// ---- FBs/B_JKS_OldFB/Memory/INDIRECT_FN.TcPOU
FUNCTION_BLOCK INDIRECT_FN
VAR_INPUT
	BOOL_SV_PB: BOOL;		(*SAVE PB (TS)*)
	BOOL_LD_PB: BOOL;			(*LOAD PB (TS)*)
	INT_P_NO: INT;		(*PROGRAM NO (TS) 1~10*)
	INT_D00:INT;
	INT_D01:INT;
	INT_D02:INT;
	INT_D03:INT;
	INT_D04:INT;
	INT_D05:INT;
	INT_D06:INT;
	INT_D07:INT;
	INT_D08:INT;
	INT_D09:INT;
	INT_D10:INT;
	INT_D11:INT;
	INT_D12:INT;
	INT_D13:INT;
	INT_D14:INT;
	INT_D15:INT;
	INT_D16:INT;
	INT_D17:INT;
	INT_D18:INT;
	INT_D19:INT;
	INT_D20:INT;
	INT_D21:INT;
	INT_D22:INT;
	INT_D23:INT;
	INT_D24:INT;
	INT_D25:INT;
	INT_D26:INT;
	INT_D27:INT;
	INT_D28:INT;
	INT_D29:INT;
	INT_D30:INT;
	STG_STG1:STRING;
END_VAR
VAR_OUTPUT
	SV_PB_IND_BOOL:BOOL;
	LD_PB_IND_BOOL:BOOL;
	D00_INT:INT;
	D01_INT:INT;
	D02_INT:INT;
	D03_INT:INT;
	D04_INT:INT;
	D05_INT:INT;
	D06_INT:INT;
	D07_INT:INT;
	D08_INT:INT;
	D09_INT:INT;
	D10_INT:INT;
	D11_INT:INT;
	D12_INT:INT;
	D13_INT:INT;
	D14_INT:INT;
	D15_INT:INT;
	D16_INT:INT;
	D17_INT:INT;
	D18_INT:INT;
	D19_INT:INT;
	D20_INT:INT;
	D21_INT:INT;
	D22_INT:INT;
	D23_INT:INT;
	D24_INT:INT;
	D25_INT:INT;
	D26_INT:INT;
	D27_INT:INT;
	D28_INT:INT;
	D29_INT:INT;
	D30_INT:INT;
	STG1_STG:STRING;
END_VAR
VAR

	P1B: BOOL;
	P2B: BOOL;
	P3B: BOOL;
	P4B: BOOL;
	P5B: BOOL;
	P6B: BOOL;
	P7B: BOOL;
	P8B: BOOL;
	P9B: BOOL;
	P10B: BOOL;
	SV_HR: BOOL;
	SV_T: TON;
	SV_CR: BOOL;
	LD_HR: BOOL;
	LD_CR: BOOL;
	LD_T: TON;
	SV_DF: R_TRIG;
	SV_PLS: BOOL;
	LD_DF: R_TRIG;
	LD_PLS: BOOL;
	ALWAYS_ON: BOOL;
	TPC: TON;
	N0: BOOL;
	TPC1: TON;
	N1: BOOL;
	CNG_P_NO: INT;
	NPC: BOOL;		(*NON PROGRAM CHANGE*)
	PCDF: R_TRIG;
	PCTDF: BOOL;
	PCDFN: F_TRIG;
	PC_PLS: BOOL;
	SVPLS: R_TRIG;
	SV_PB_PLS: BOOL;
	LDPLS: R_TRIG;
	LD_PB_PLS: BOOL;
END_VAR
VAR PERSISTENT
	P01D00:INT;
	P01D01:INT;
	P01D02:INT;
	P01D03:INT;
	P01D04:INT;
	P01D05:INT;
	P01D06:INT;
	P01D07:INT;
	P01D08:INT;
	P01D09:INT;
	P01D10:INT;
	P01D11:INT;
	P01D12:INT;
	P01D13:INT;
	P01D14:INT;
	P01D15:INT;
	P01D16:INT;
	P01D17:INT;
	P01D18:INT;
	P01D19:INT;
	P01D20:INT;
	P01D21:INT;
	P01D22:INT;
	P01D23:INT;
	P01D24:INT;
	P01D25:INT;
	P01D26:INT;
	P01D27:INT;
	P01D28:INT;
	P01D29:INT;
	P01D30:INT;
	P01STG:STRING;
	P02D00:INT;
	P02D01:INT;
	P02D02:INT;
	P02D03:INT;
	P02D04:INT;
	P02D05:INT;
	P02D06:INT;
	P02D07:INT;
	P02D08:INT;
	P02D09:INT;
	P02D10:INT;
	P02D11:INT;
	P02D12:INT;
	P02D13:INT;
	P02D14:INT;
	P02D15:INT;
	P02D16:INT;
	P02D17:INT;
	P02D18:INT;
	P02D19:INT;
	P02D20:INT;
	P02D21:INT;
	P02D22:INT;
	P02D23:INT;
	P02D24:INT;
	P02D25:INT;
	P02D26:INT;
	P02D27:INT;
	P02D28:INT;
	P02D29:INT;
	P02D30:INT;
	P02STG:STRING;
	P03D00:INT;
	P03D01:INT;
	P03D02:INT;
	P03D03:INT;
	P03D04:INT;
	P03D05:INT;
	P03D06:INT;
	P03D07:INT;
	P03D08:INT;
	P03D09:INT;
	P03D10:INT;
	P03D11:INT;
	P03D12:INT;
	P03D13:INT;
	P03D14:INT;
	P03D15:INT;
	P03D16:INT;
	P03D17:INT;
	P03D18:INT;
	P03D19:INT;
	P03D20:INT;
	P03D21:INT;
	P03D22:INT;
	P03D23:INT;
	P03D24:INT;
	P03D25:INT;
	P03D26:INT;
	P03D27:INT;
	P03D28:INT;
	P03D29:INT;
	P03D30:INT;
	P03STG:STRING;
	P04D00:INT;
	P04D01:INT;
	P04D02:INT;
	P04D03:INT;
	P04D04:INT;
	P04D05:INT;
	P04D06:INT;
	P04D07:INT;
	P04D08:INT;
	P04D09:INT;
	P04D10:INT;
	P04D11:INT;
	P04D12:INT;
	P04D13:INT;
	P04D14:INT;
	P04D15:INT;
	P04D16:INT;
	P04D17:INT;
	P04D18:INT;
	P04D19:INT;
	P04D20:INT;
	P04D21:INT;
	P04D22:INT;
	P04D23:INT;
	P04D24:INT;
	P04D25:INT;
	P04D26:INT;
	P04D27:INT;
	P04D28:INT;
	P04D29:INT;
	P04D30:INT;
	P04STG:STRING;
	P05D00:INT;
	P05D01:INT;
	P05D02:INT;
	P05D03:INT;
	P05D04:INT;
	P05D05:INT;
	P05D06:INT;
	P05D07:INT;
	P05D08:INT;
	P05D09:INT;
	P05D10:INT;
	P05D11:INT;
	P05D12:INT;
	P05D13:INT;
	P05D14:INT;
	P05D15:INT;
	P05D16:INT;
	P05D17:INT;
	P05D18:INT;
	P05D19:INT;
	P05D20:INT;
	P05D21:INT;
	P05D22:INT;
	P05D23:INT;
	P05D24:INT;
	P05D25:INT;
	P05D26:INT;
	P05D27:INT;
	P05D28:INT;
	P05D29:INT;
	P05D30:INT;
	P05STG:STRING;
	P06D00:INT;
	P06D01:INT;
	P06D02:INT;
	P06D03:INT;
	P06D04:INT;
	P06D05:INT;
	P06D06:INT;
	P06D07:INT;
	P06D08:INT;
	P06D09:INT;
	P06D10:INT;
	P06D11:INT;
	P06D12:INT;
	P06D13:INT;
	P06D14:INT;
	P06D15:INT;
	P06D16:INT;
	P06D17:INT;
	P06D18:INT;
	P06D19:INT;
	P06D20:INT;
	P06D21:INT;
	P06D22:INT;
	P06D23:INT;
	P06D24:INT;
	P06D25:INT;
	P06D26:INT;
	P06D27:INT;
	P06D28:INT;
	P06D29:INT;
	P06D30:INT;
	P06STG:STRING;
	P07D00:INT;
	P07D01:INT;
	P07D02:INT;
	P07D03:INT;
	P07D04:INT;
	P07D05:INT;
	P07D06:INT;
	P07D07:INT;
	P07D08:INT;
	P07D09:INT;
	P07D10:INT;
	P07D11:INT;
	P07D12:INT;
	P07D13:INT;
	P07D14:INT;
	P07D15:INT;
	P07D16:INT;
	P07D17:INT;
	P07D18:INT;
	P07D19:INT;
	P07D20:INT;
	P07D21:INT;
	P07D22:INT;
	P07D23:INT;
	P07D24:INT;
	P07D25:INT;
	P07D26:INT;
	P07D27:INT;
	P07D28:INT;
	P07D29:INT;
	P07D30:INT;
	P07STG:STRING;
	P08D00:INT;
	P08D01:INT;
	P08D02:INT;
	P08D03:INT;
	P08D04:INT;
	P08D05:INT;
	P08D06:INT;
	P08D07:INT;
	P08D08:INT;
	P08D09:INT;
	P08D10:INT;
	P08D11:INT;
	P08D12:INT;
	P08D13:INT;
	P08D14:INT;
	P08D15:INT;
	P08D16:INT;
	P08D17:INT;
	P08D18:INT;
	P08D19:INT;
	P08D20:INT;
	P08D21:INT;
	P08D22:INT;
	P08D23:INT;
	P08D24:INT;
	P08D25:INT;
	P08D26:INT;
	P08D27:INT;
	P08D28:INT;
	P08D29:INT;
	P08D30:INT;
	P08STG:STRING;
	P09D00:INT;
	P09D01:INT;
	P09D02:INT;
	P09D03:INT;
	P09D04:INT;
	P09D05:INT;
	P09D06:INT;
	P09D07:INT;
	P09D08:INT;
	P09D09:INT;
	P09D10:INT;
	P09D11:INT;
	P09D12:INT;
	P09D13:INT;
	P09D14:INT;
	P09D15:INT;
	P09D16:INT;
	P09D17:INT;
	P09D18:INT;
	P09D19:INT;
	P09D20:INT;
	P09D21:INT;
	P09D22:INT;
	P09D23:INT;
	P09D24:INT;
	P09D25:INT;
	P09D26:INT;
	P09D27:INT;
	P09D28:INT;
	P09D29:INT;
	P09D30:INT;
	P09STG:STRING;
	P10D00:INT;
	P10D01:INT;
	P10D02:INT;
	P10D03:INT;
	P10D04:INT;
	P10D05:INT;
	P10D06:INT;
	P10D07:INT;
	P10D08:INT;
	P10D09:INT;
	P10D10:INT;
	P10D11:INT;
	P10D12:INT;
	P10D13:INT;
	P10D14:INT;
	P10D15:INT;
	P10D16:INT;
	P10D17:INT;
	P10D18:INT;
	P10D19:INT;
	P10D20:INT;
	P10D21:INT;
	P10D22:INT;
	P10D23:INT;
	P10D24:INT;
	P10D25:INT;
	P10D26:INT;
	P10D27:INT;
	P10D28:INT;
	P10D29:INT;
	P10D30:INT;
	P10STG:STRING;

END_VAR
VAR // added by the converter: edge detectors and wires of the graphical bodies
    _w1, _w35, _w68, _w101, _w134, _w167, _w200, _w233, _w266, _w299, _w332, _w365, _w398, _w431, _w464, _w497, _w530, _w563, _w596, _w629, _w662 : BOOL;
    _w2, _w3, _w4, _w5, _w6, _w7, _w8, _w9, _w10, _w11, _w12, _w13, _w14, _w15, _w16, _w17, _w18, _w19, _w20, _w21, _w22, _w23, _w24, _w25, _w26, _w27, _w28, _w29, _w30, _w31, _w32, _w34, _w36, _w37, _w38, _w39, _w40, _w41, _w42, _w43, _w44, _w45, _w46, _w47, _w48, _w49, _w50, _w51, _w52, _w53, _w54, _w55, _w56, _w57, _w58, _w59, _w60, _w61, _w62, _w63, _w64, _w65, _w66, _w69, _w70, _w71, _w72, _w73, _w74, _w75, _w76, _w77, _w78, _w79, _w80, _w81, _w82, _w83, _w84, _w85, _w86, _w87, _w88, _w89, _w90, _w91, _w92, _w93, _w94, _w95, _w96, _w97, _w98, _w99, _w102, _w103, _w104, _w105, _w106, _w107, _w108, _w109, _w110, _w111, _w112, _w113, _w114, _w115, _w116, _w117, _w118, _w119, _w120, _w121, _w122, _w123, _w124, _w125, _w126, _w127, _w128, _w129, _w130, _w131, _w132, _w135, _w136, _w137, _w138, _w139, _w140, _w141, _w142, _w143, _w144, _w145, _w146, _w147, _w148, _w149, _w150, _w151, _w152, _w153, _w154, _w155, _w156, _w157, _w158, _w159, _w160, _w161, _w162, _w163, _w164, _w165, _w168, _w169, _w170, _w171, _w172, _w173, _w174, _w175, _w176, _w177, _w178, _w179, _w180, _w181, _w182, _w183, _w184, _w185, _w186, _w187, _w188, _w189, _w190, _w191, _w192, _w193, _w194, _w195, _w196, _w197, _w198, _w201, _w202, _w203, _w204, _w205, _w206, _w207, _w208, _w209, _w210, _w211, _w212, _w213, _w214, _w215, _w216, _w217, _w218, _w219, _w220, _w221, _w222, _w223, _w224, _w225, _w226, _w227, _w228, _w229, _w230, _w231, _w234, _w235, _w236, _w237, _w238, _w239, _w240, _w241, _w242, _w243, _w244, _w245, _w246, _w247, _w248, _w249, _w250, _w251, _w252, _w253, _w254, _w255, _w256, _w257, _w258, _w259, _w260, _w261, _w262, _w263, _w264, _w267, _w268, _w269, _w270, _w271, _w272, _w273, _w274, _w275, _w276, _w277, _w278, _w279, _w280, _w281, _w282, _w283, _w284, _w285, _w286, _w287, _w288, _w289, _w290, _w291, _w292, _w293, _w294, _w295, _w296, _w297, _w300, _w301, _w302, _w303, _w304, _w305, _w306, _w307, _w308, _w309, _w310, _w311, _w312, _w313, _w314, _w315, _w316, _w317, _w318, _w319, _w320, _w321, _w322, _w323, _w324, _w325, _w326, _w327, _w328, _w329, _w330, _w333, _w334, _w335, _w336, _w337, _w338, _w339, _w340, _w341, _w342, _w343, _w344, _w345, _w346, _w347, _w348, _w349, _w350, _w351, _w352, _w353, _w354, _w355, _w356, _w357, _w358, _w359, _w360, _w361, _w362, _w363, _w366, _w367, _w368, _w369, _w370, _w371, _w372, _w373, _w374, _w375, _w376, _w377, _w378, _w379, _w380, _w381, _w382, _w383, _w384, _w385, _w386, _w387, _w388, _w389, _w390, _w391, _w392, _w393, _w394, _w395, _w396, _w399, _w400, _w401, _w402, _w403, _w404, _w405, _w406, _w407, _w408, _w409, _w410, _w411, _w412, _w413, _w414, _w415, _w416, _w417, _w418, _w419, _w420, _w421, _w422, _w423, _w424, _w425, _w426, _w427, _w428, _w429, _w432, _w433, _w434, _w435, _w436, _w437, _w438, _w439, _w440, _w441, _w442, _w443, _w444, _w445, _w446, _w447, _w448, _w449, _w450, _w451, _w452, _w453, _w454, _w455, _w456, _w457, _w458, _w459, _w460, _w461, _w462, _w465, _w466, _w467, _w468, _w469, _w470, _w471, _w472, _w473, _w474, _w475, _w476, _w477, _w478, _w479, _w480, _w481, _w482, _w483, _w484, _w485, _w486, _w487, _w488, _w489, _w490, _w491, _w492, _w493, _w494, _w495, _w498, _w499, _w500, _w501, _w502, _w503, _w504, _w505, _w506, _w507, _w508, _w509, _w510, _w511, _w512, _w513, _w514, _w515, _w516, _w517, _w518, _w519, _w520, _w521, _w522, _w523, _w524, _w525, _w526, _w527, _w528, _w531, _w532, _w533, _w534, _w535, _w536, _w537, _w538, _w539, _w540, _w541, _w542, _w543, _w544, _w545, _w546, _w547, _w548, _w549, _w550, _w551, _w552, _w553, _w554, _w555, _w556, _w557, _w558, _w559, _w560, _w561, _w564, _w565, _w566, _w567, _w568, _w569, _w570, _w571, _w572, _w573, _w574, _w575, _w576, _w577, _w578, _w579, _w580, _w581, _w582, _w583, _w584, _w585, _w586, _w587, _w588, _w589, _w590, _w591, _w592, _w593, _w594, _w597, _w598, _w599, _w600, _w601, _w602, _w603, _w604, _w605, _w606, _w607, _w608, _w609, _w610, _w611, _w612, _w613, _w614, _w615, _w616, _w617, _w618, _w619, _w620, _w621, _w622, _w623, _w624, _w625, _w626, _w627, _w630, _w631, _w632, _w633, _w634, _w635, _w636, _w637, _w638, _w639, _w640, _w641, _w642, _w643, _w644, _w645, _w646, _w647, _w648, _w649, _w650, _w651, _w652, _w653, _w654, _w655, _w656, _w657, _w658, _w659, _w660, _w663, _w664, _w665, _w666, _w667, _w668, _w669, _w670, _w671, _w672, _w673, _w674, _w675, _w676, _w677, _w678, _w679, _w680, _w681, _w682, _w683, _w684, _w685, _w686, _w687, _w688, _w689, _w690, _w691, _w692, _w693 : INT;
    _w33, _w67, _w100, _w133, _w166, _w199, _w232, _w265, _w298, _w331, _w364, _w397, _w430, _w463, _w496, _w529, _w562, _w595, _w628, _w661, _w694 : STRING;
END_VAR

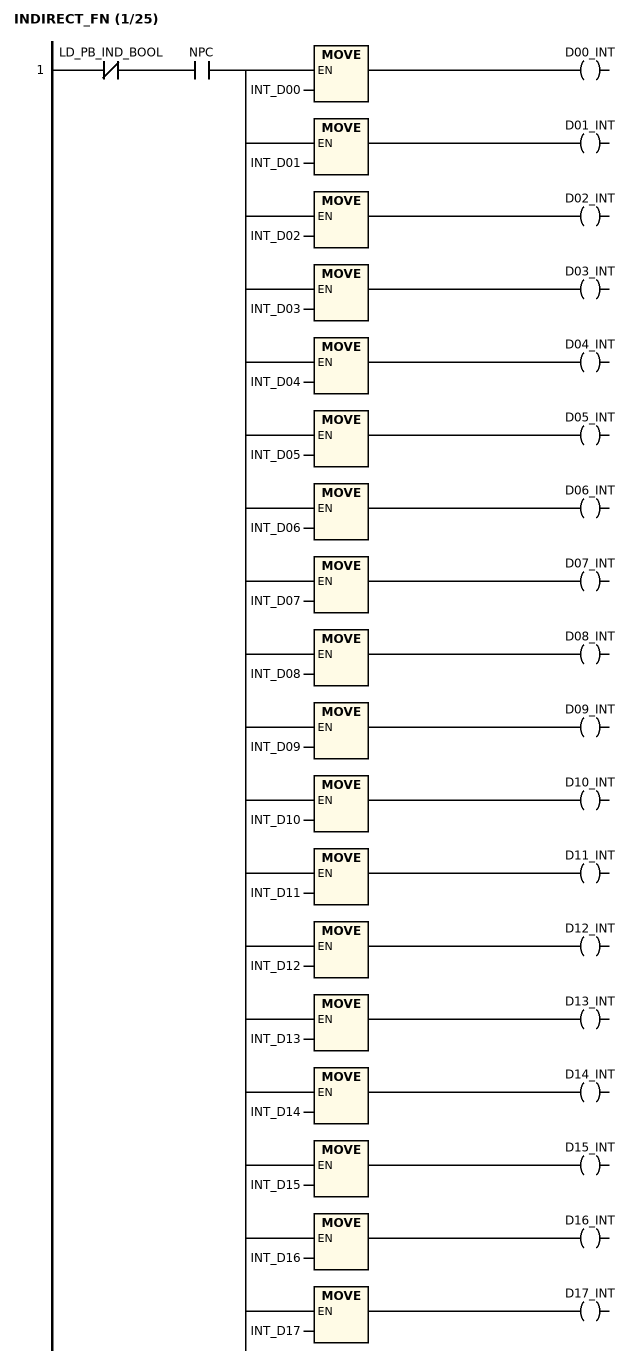
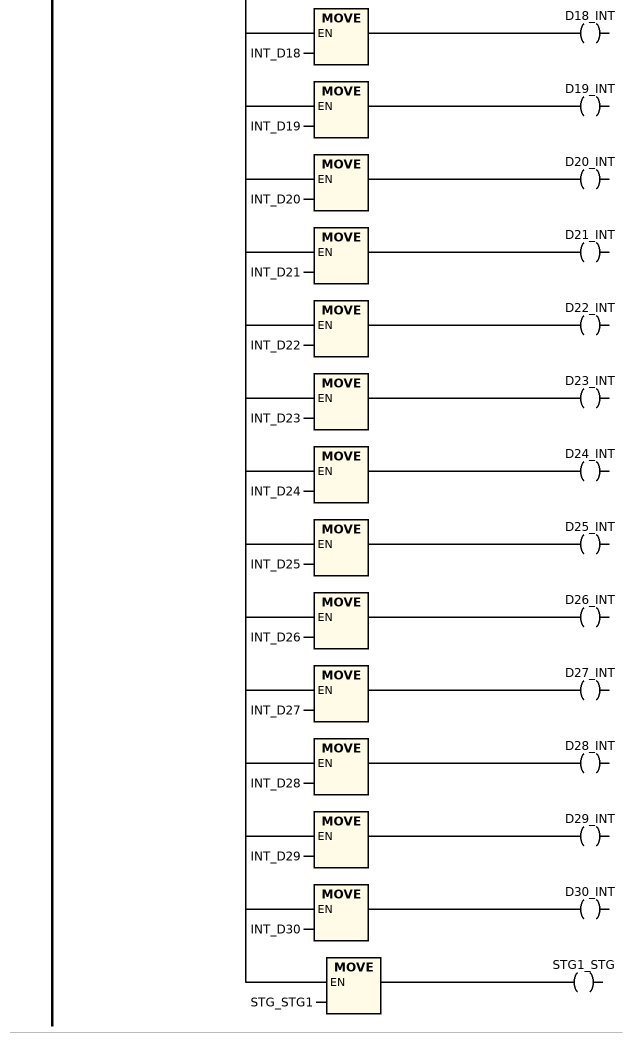
// NETWORK 1
_w1 := NOT LD_PB_IND_BOOL AND NPC;
IF _w1 THEN _w2 := INT_D00; END_IF
D00_INT := _w2;
IF _w1 THEN _w3 := INT_D01; END_IF
D01_INT := _w3;
IF _w1 THEN _w4 := INT_D02; END_IF
D02_INT := _w4;
IF _w1 THEN _w5 := INT_D03; END_IF
D03_INT := _w5;
IF _w1 THEN _w6 := INT_D04; END_IF
D04_INT := _w6;
IF _w1 THEN _w7 := INT_D05; END_IF
D05_INT := _w7;
IF _w1 THEN _w8 := INT_D06; END_IF
D06_INT := _w8;
IF _w1 THEN _w9 := INT_D07; END_IF
D07_INT := _w9;
IF _w1 THEN _w10 := INT_D08; END_IF
D08_INT := _w10;
IF _w1 THEN _w11 := INT_D09; END_IF
D09_INT := _w11;
IF _w1 THEN _w12 := INT_D10; END_IF
D10_INT := _w12;
IF _w1 THEN _w13 := INT_D11; END_IF
D11_INT := _w13;
IF _w1 THEN _w14 := INT_D12; END_IF
D12_INT := _w14;
IF _w1 THEN _w15 := INT_D13; END_IF
D13_INT := _w15;
IF _w1 THEN _w16 := INT_D14; END_IF
D14_INT := _w16;
IF _w1 THEN _w17 := INT_D15; END_IF
D15_INT := _w17;
IF _w1 THEN _w18 := INT_D16; END_IF
D16_INT := _w18;
IF _w1 THEN _w19 := INT_D17; END_IF
D17_INT := _w19;
IF _w1 THEN _w20 := INT_D18; END_IF
D18_INT := _w20;
IF _w1 THEN _w21 := INT_D19; END_IF
D19_INT := _w21;
IF _w1 THEN _w22 := INT_D20; END_IF
D20_INT := _w22;
IF _w1 THEN _w23 := INT_D21; END_IF
D21_INT := _w23;
IF _w1 THEN _w24 := INT_D22; END_IF
D22_INT := _w24;
IF _w1 THEN _w25 := INT_D23; END_IF
D23_INT := _w25;
IF _w1 THEN _w26 := INT_D24; END_IF
D24_INT := _w26;
IF _w1 THEN _w27 := INT_D25; END_IF
D25_INT := _w27;
IF _w1 THEN _w28 := INT_D26; END_IF
D26_INT := _w28;
IF _w1 THEN _w29 := INT_D27; END_IF
D27_INT := _w29;
IF _w1 THEN _w30 := INT_D28; END_IF
D28_INT := _w30;
IF _w1 THEN _w31 := INT_D29; END_IF
D29_INT := _w31;
IF _w1 THEN _w32 := INT_D30; END_IF
D30_INT := _w32;
IF _w1 THEN _w33 := STG_STG1; END_IF
STG1_STG := _w33;

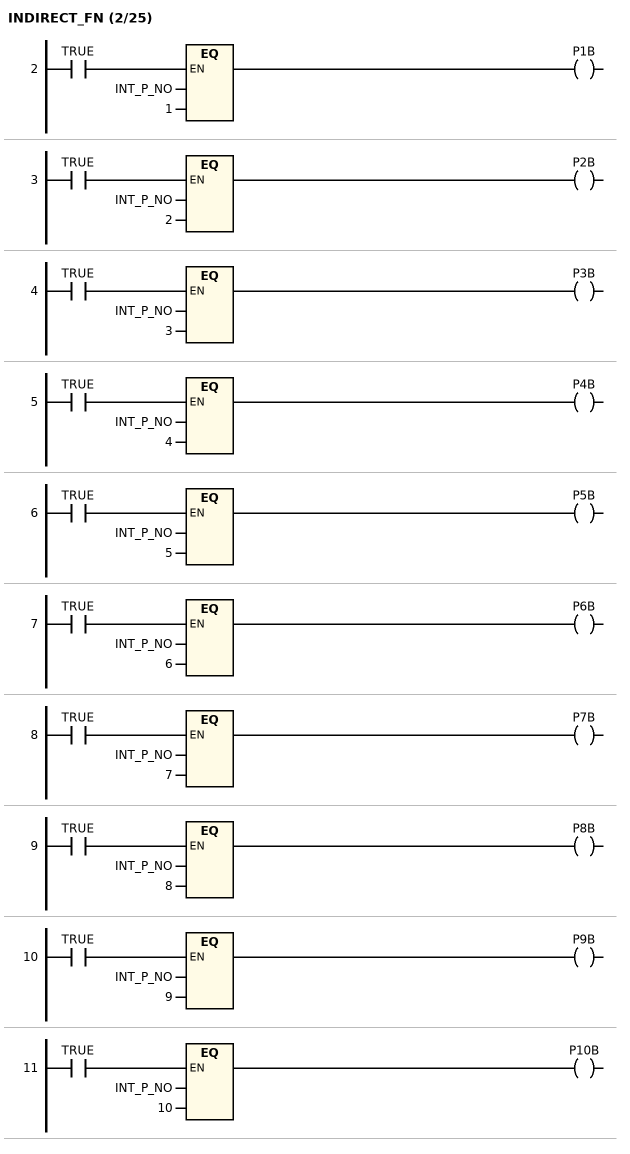
// NETWORK 2
P1B := INT_P_NO = 1;

// NETWORK 3
P2B := INT_P_NO = 2;

// NETWORK 4
P3B := INT_P_NO = 3;

// NETWORK 5
P4B := INT_P_NO = 4;

// NETWORK 6
P5B := INT_P_NO = 5;

// NETWORK 7
P6B := INT_P_NO = 6;

// NETWORK 8
P7B := INT_P_NO = 7;

// NETWORK 9
P8B := INT_P_NO = 8;

// NETWORK 10
P9B := INT_P_NO = 9;

// NETWORK 11
P10B := INT_P_NO = 10;

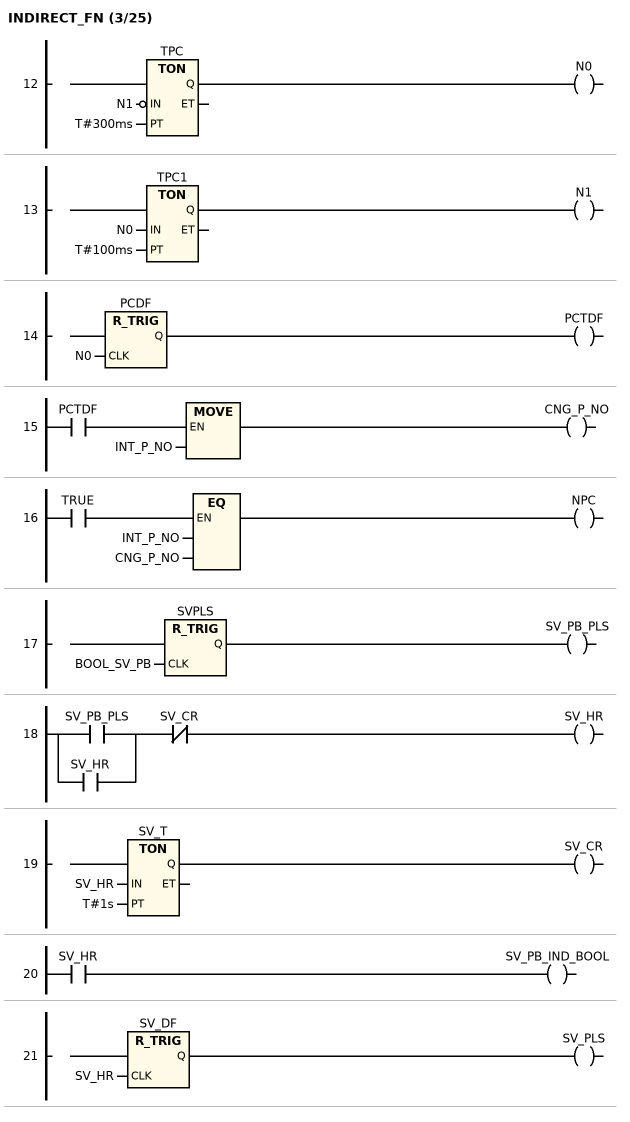
// NETWORK 12
TPC(IN := NOT N1, PT := T#300ms); // TON
N0 := TPC.Q;

// NETWORK 13
TPC1(IN := N0, PT := T#100ms); // TON
N1 := TPC1.Q;

// NETWORK 14
PCDF(CLK := N0); // R_TRIG
PCTDF := PCDF.Q;

// NETWORK 15
IF PCTDF THEN _w34 := INT_P_NO; END_IF
CNG_P_NO := _w34;

// NETWORK 16
NPC := INT_P_NO = CNG_P_NO;

// NETWORK 17
SVPLS(CLK := BOOL_SV_PB); // R_TRIG
SV_PB_PLS := SVPLS.Q;

// NETWORK 18
SV_HR := (SV_PB_PLS OR SV_HR) AND NOT SV_CR;

// NETWORK 19
SV_T(IN := SV_HR, PT := T#1s); // TON
SV_CR := SV_T.Q;

// NETWORK 20
SV_PB_IND_BOOL := SV_HR;

// NETWORK 21
SV_DF(CLK := SV_HR); // R_TRIG
SV_PLS := SV_DF.Q;

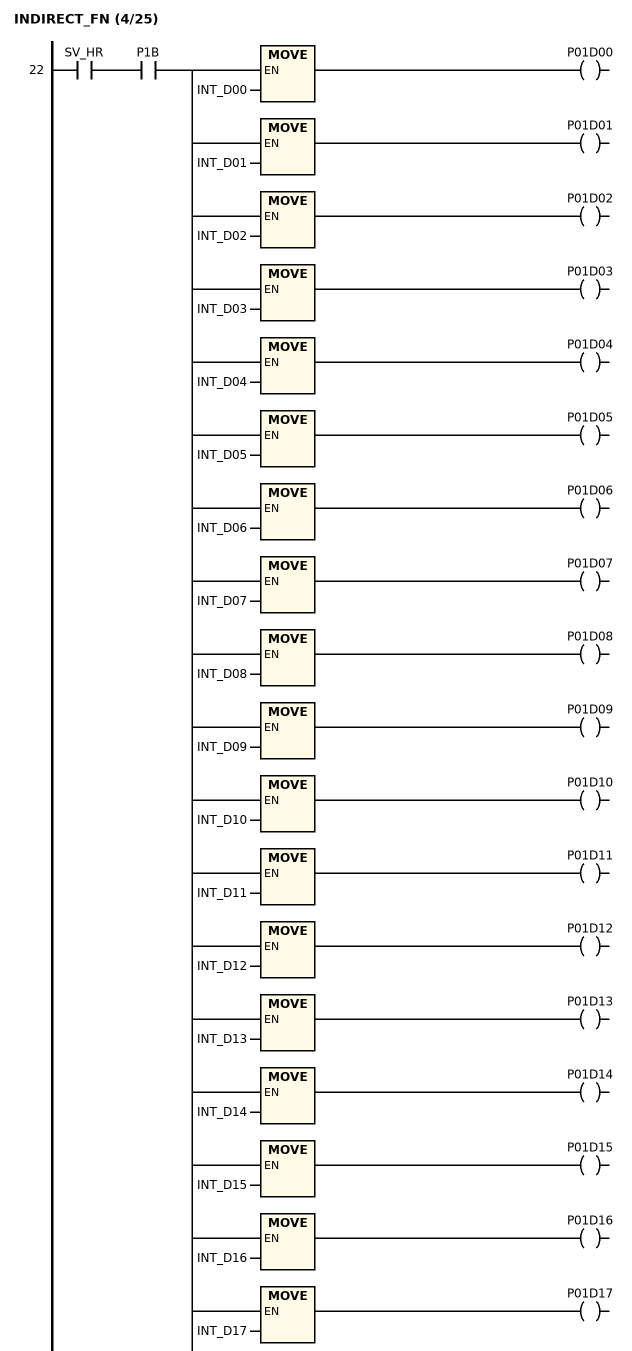
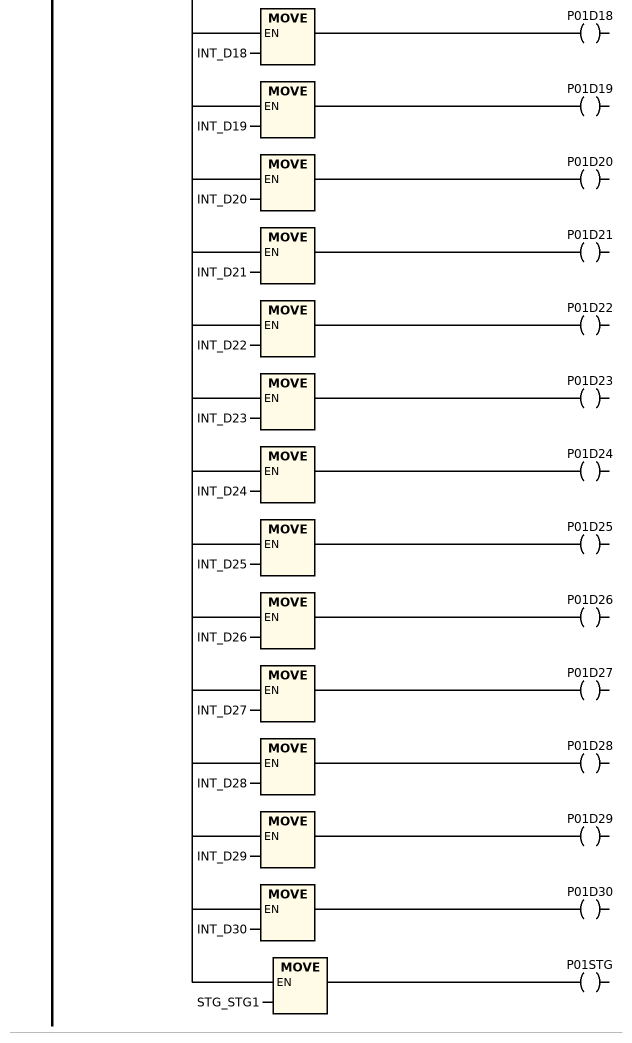
// NETWORK 22
_w35 := SV_HR AND P1B;
IF _w35 THEN _w36 := INT_D00; END_IF
P01D00 := _w36;
IF _w35 THEN _w37 := INT_D01; END_IF
P01D01 := _w37;
IF _w35 THEN _w38 := INT_D02; END_IF
P01D02 := _w38;
IF _w35 THEN _w39 := INT_D03; END_IF
P01D03 := _w39;
IF _w35 THEN _w40 := INT_D04; END_IF
P01D04 := _w40;
IF _w35 THEN _w41 := INT_D05; END_IF
P01D05 := _w41;
IF _w35 THEN _w42 := INT_D06; END_IF
P01D06 := _w42;
IF _w35 THEN _w43 := INT_D07; END_IF
P01D07 := _w43;
IF _w35 THEN _w44 := INT_D08; END_IF
P01D08 := _w44;
IF _w35 THEN _w45 := INT_D09; END_IF
P01D09 := _w45;
IF _w35 THEN _w46 := INT_D10; END_IF
P01D10 := _w46;
IF _w35 THEN _w47 := INT_D11; END_IF
P01D11 := _w47;
IF _w35 THEN _w48 := INT_D12; END_IF
P01D12 := _w48;
IF _w35 THEN _w49 := INT_D13; END_IF
P01D13 := _w49;
IF _w35 THEN _w50 := INT_D14; END_IF
P01D14 := _w50;
IF _w35 THEN _w51 := INT_D15; END_IF
P01D15 := _w51;
IF _w35 THEN _w52 := INT_D16; END_IF
P01D16 := _w52;
IF _w35 THEN _w53 := INT_D17; END_IF
P01D17 := _w53;
IF _w35 THEN _w54 := INT_D18; END_IF
P01D18 := _w54;
IF _w35 THEN _w55 := INT_D19; END_IF
P01D19 := _w55;
IF _w35 THEN _w56 := INT_D20; END_IF
P01D20 := _w56;
IF _w35 THEN _w57 := INT_D21; END_IF
P01D21 := _w57;
IF _w35 THEN _w58 := INT_D22; END_IF
P01D22 := _w58;
IF _w35 THEN _w59 := INT_D23; END_IF
P01D23 := _w59;
IF _w35 THEN _w60 := INT_D24; END_IF
P01D24 := _w60;
IF _w35 THEN _w61 := INT_D25; END_IF
P01D25 := _w61;
IF _w35 THEN _w62 := INT_D26; END_IF
P01D26 := _w62;
IF _w35 THEN _w63 := INT_D27; END_IF
P01D27 := _w63;
IF _w35 THEN _w64 := INT_D28; END_IF
P01D28 := _w64;
IF _w35 THEN _w65 := INT_D29; END_IF
P01D29 := _w65;
IF _w35 THEN _w66 := INT_D30; END_IF
P01D30 := _w66;
IF _w35 THEN _w67 := STG_STG1; END_IF
P01STG := _w67;

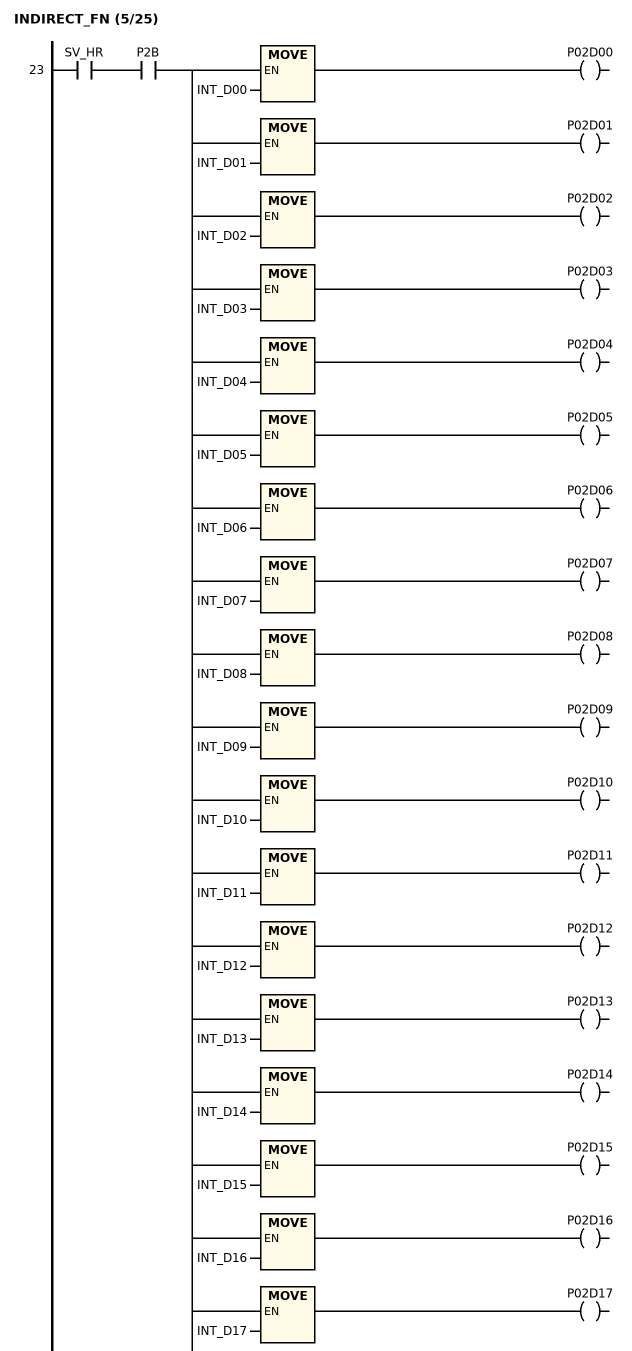
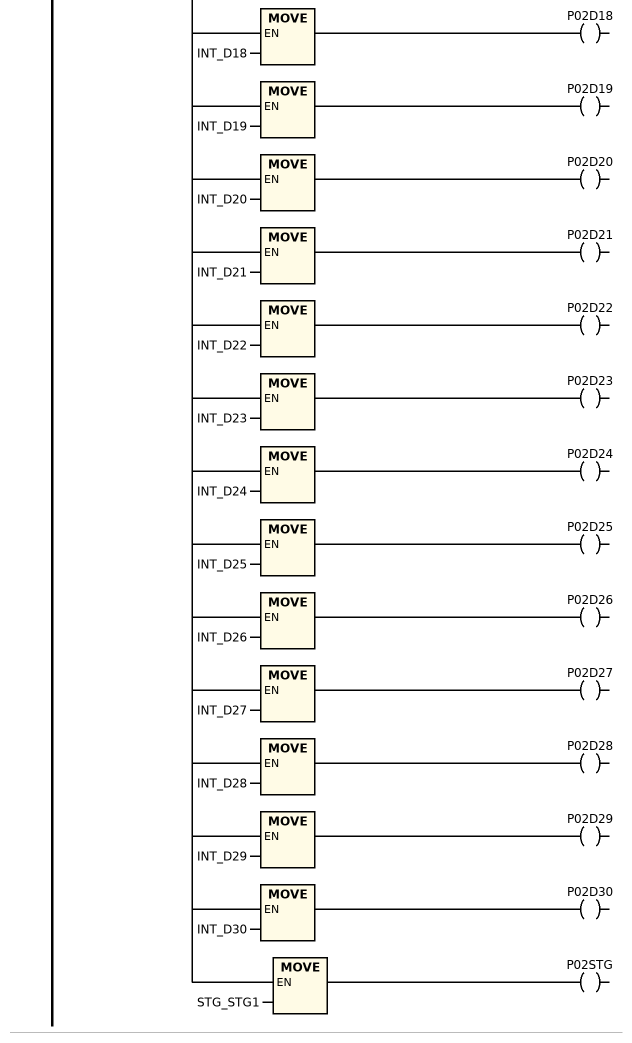
// NETWORK 23
_w68 := SV_HR AND P2B;
IF _w68 THEN _w69 := INT_D00; END_IF
P02D00 := _w69;
IF _w68 THEN _w70 := INT_D01; END_IF
P02D01 := _w70;
IF _w68 THEN _w71 := INT_D02; END_IF
P02D02 := _w71;
IF _w68 THEN _w72 := INT_D03; END_IF
P02D03 := _w72;
IF _w68 THEN _w73 := INT_D04; END_IF
P02D04 := _w73;
IF _w68 THEN _w74 := INT_D05; END_IF
P02D05 := _w74;
IF _w68 THEN _w75 := INT_D06; END_IF
P02D06 := _w75;
IF _w68 THEN _w76 := INT_D07; END_IF
P02D07 := _w76;
IF _w68 THEN _w77 := INT_D08; END_IF
P02D08 := _w77;
IF _w68 THEN _w78 := INT_D09; END_IF
P02D09 := _w78;
IF _w68 THEN _w79 := INT_D10; END_IF
P02D10 := _w79;
IF _w68 THEN _w80 := INT_D11; END_IF
P02D11 := _w80;
IF _w68 THEN _w81 := INT_D12; END_IF
P02D12 := _w81;
IF _w68 THEN _w82 := INT_D13; END_IF
P02D13 := _w82;
IF _w68 THEN _w83 := INT_D14; END_IF
P02D14 := _w83;
IF _w68 THEN _w84 := INT_D15; END_IF
P02D15 := _w84;
IF _w68 THEN _w85 := INT_D16; END_IF
P02D16 := _w85;
IF _w68 THEN _w86 := INT_D17; END_IF
P02D17 := _w86;
IF _w68 THEN _w87 := INT_D18; END_IF
P02D18 := _w87;
IF _w68 THEN _w88 := INT_D19; END_IF
P02D19 := _w88;
IF _w68 THEN _w89 := INT_D20; END_IF
P02D20 := _w89;
IF _w68 THEN _w90 := INT_D21; END_IF
P02D21 := _w90;
IF _w68 THEN _w91 := INT_D22; END_IF
P02D22 := _w91;
IF _w68 THEN _w92 := INT_D23; END_IF
P02D23 := _w92;
IF _w68 THEN _w93 := INT_D24; END_IF
P02D24 := _w93;
IF _w68 THEN _w94 := INT_D25; END_IF
P02D25 := _w94;
IF _w68 THEN _w95 := INT_D26; END_IF
P02D26 := _w95;
IF _w68 THEN _w96 := INT_D27; END_IF
P02D27 := _w96;
IF _w68 THEN _w97 := INT_D28; END_IF
P02D28 := _w97;
IF _w68 THEN _w98 := INT_D29; END_IF
P02D29 := _w98;
IF _w68 THEN _w99 := INT_D30; END_IF
P02D30 := _w99;
IF _w68 THEN _w100 := STG_STG1; END_IF
P02STG := _w100;

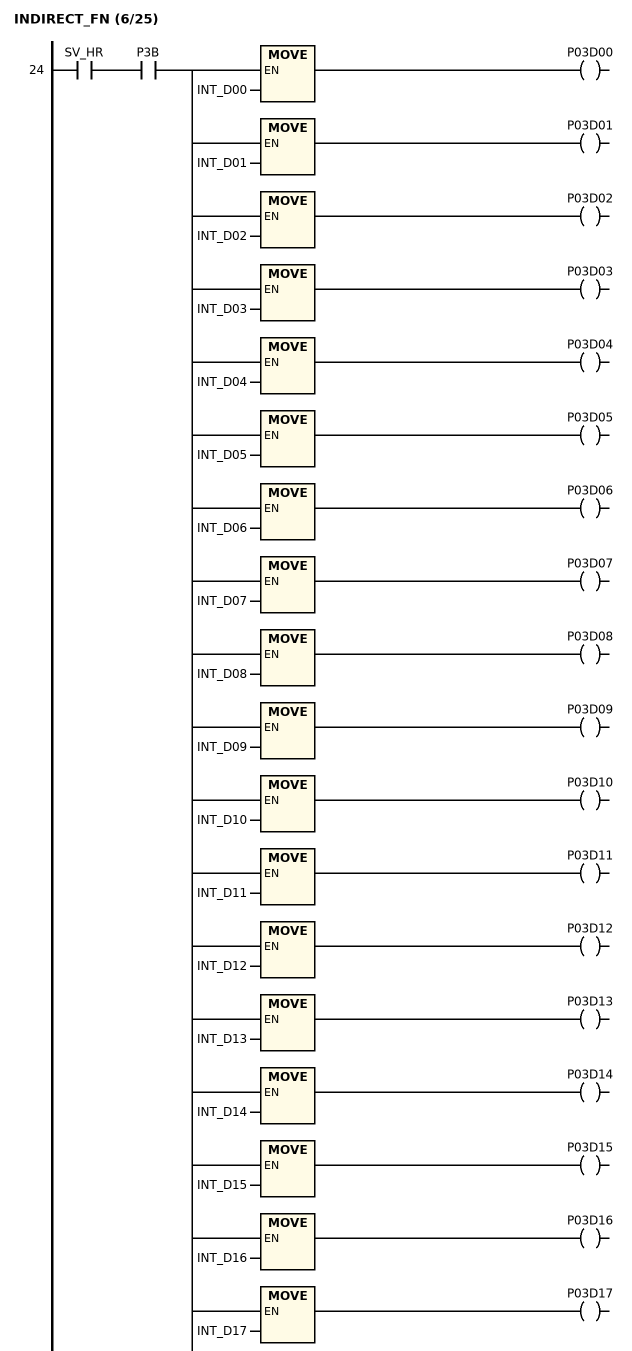
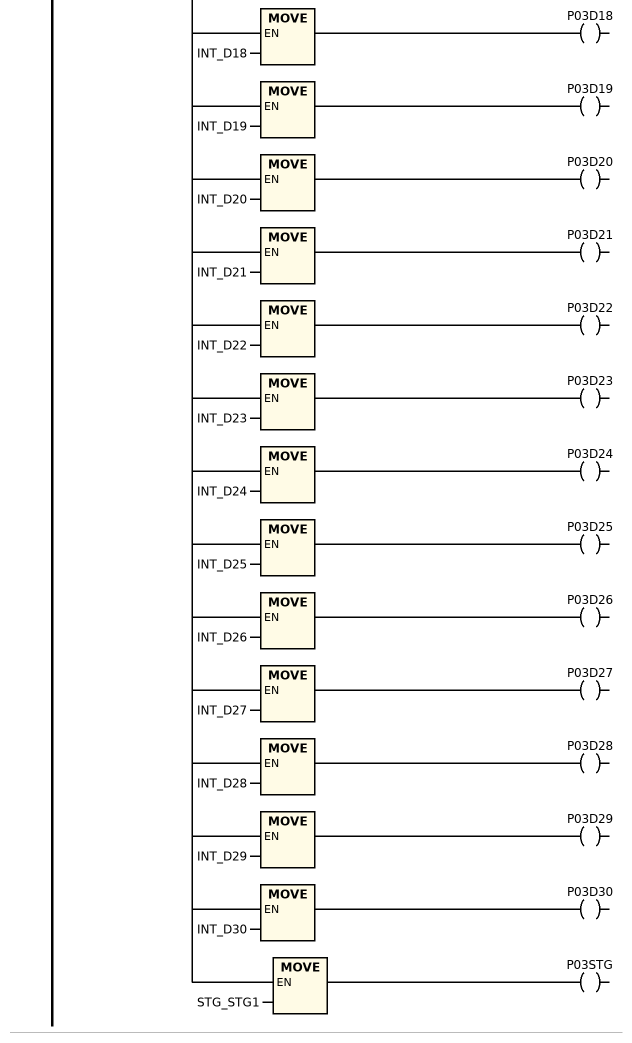
// NETWORK 24
_w101 := SV_HR AND P3B;
IF _w101 THEN _w102 := INT_D00; END_IF
P03D00 := _w102;
IF _w101 THEN _w103 := INT_D01; END_IF
P03D01 := _w103;
IF _w101 THEN _w104 := INT_D02; END_IF
P03D02 := _w104;
IF _w101 THEN _w105 := INT_D03; END_IF
P03D03 := _w105;
IF _w101 THEN _w106 := INT_D04; END_IF
P03D04 := _w106;
IF _w101 THEN _w107 := INT_D05; END_IF
P03D05 := _w107;
IF _w101 THEN _w108 := INT_D06; END_IF
P03D06 := _w108;
IF _w101 THEN _w109 := INT_D07; END_IF
P03D07 := _w109;
IF _w101 THEN _w110 := INT_D08; END_IF
P03D08 := _w110;
IF _w101 THEN _w111 := INT_D09; END_IF
P03D09 := _w111;
IF _w101 THEN _w112 := INT_D10; END_IF
P03D10 := _w112;
IF _w101 THEN _w113 := INT_D11; END_IF
P03D11 := _w113;
IF _w101 THEN _w114 := INT_D12; END_IF
P03D12 := _w114;
IF _w101 THEN _w115 := INT_D13; END_IF
P03D13 := _w115;
IF _w101 THEN _w116 := INT_D14; END_IF
P03D14 := _w116;
IF _w101 THEN _w117 := INT_D15; END_IF
P03D15 := _w117;
IF _w101 THEN _w118 := INT_D16; END_IF
P03D16 := _w118;
IF _w101 THEN _w119 := INT_D17; END_IF
P03D17 := _w119;
IF _w101 THEN _w120 := INT_D18; END_IF
P03D18 := _w120;
IF _w101 THEN _w121 := INT_D19; END_IF
P03D19 := _w121;
IF _w101 THEN _w122 := INT_D20; END_IF
P03D20 := _w122;
IF _w101 THEN _w123 := INT_D21; END_IF
P03D21 := _w123;
IF _w101 THEN _w124 := INT_D22; END_IF
P03D22 := _w124;
IF _w101 THEN _w125 := INT_D23; END_IF
P03D23 := _w125;
IF _w101 THEN _w126 := INT_D24; END_IF
P03D24 := _w126;
IF _w101 THEN _w127 := INT_D25; END_IF
P03D25 := _w127;
IF _w101 THEN _w128 := INT_D26; END_IF
P03D26 := _w128;
IF _w101 THEN _w129 := INT_D27; END_IF
P03D27 := _w129;
IF _w101 THEN _w130 := INT_D28; END_IF
P03D28 := _w130;
IF _w101 THEN _w131 := INT_D29; END_IF
P03D29 := _w131;
IF _w101 THEN _w132 := INT_D30; END_IF
P03D30 := _w132;
IF _w101 THEN _w133 := STG_STG1; END_IF
P03STG := _w133;

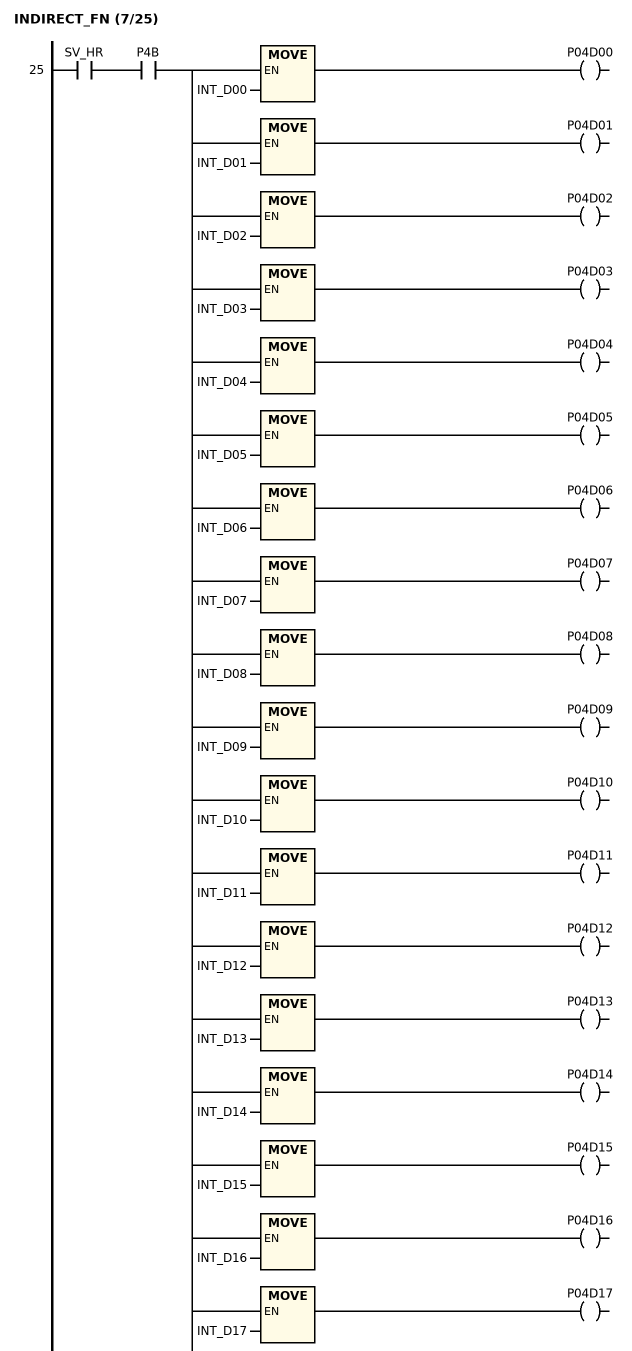
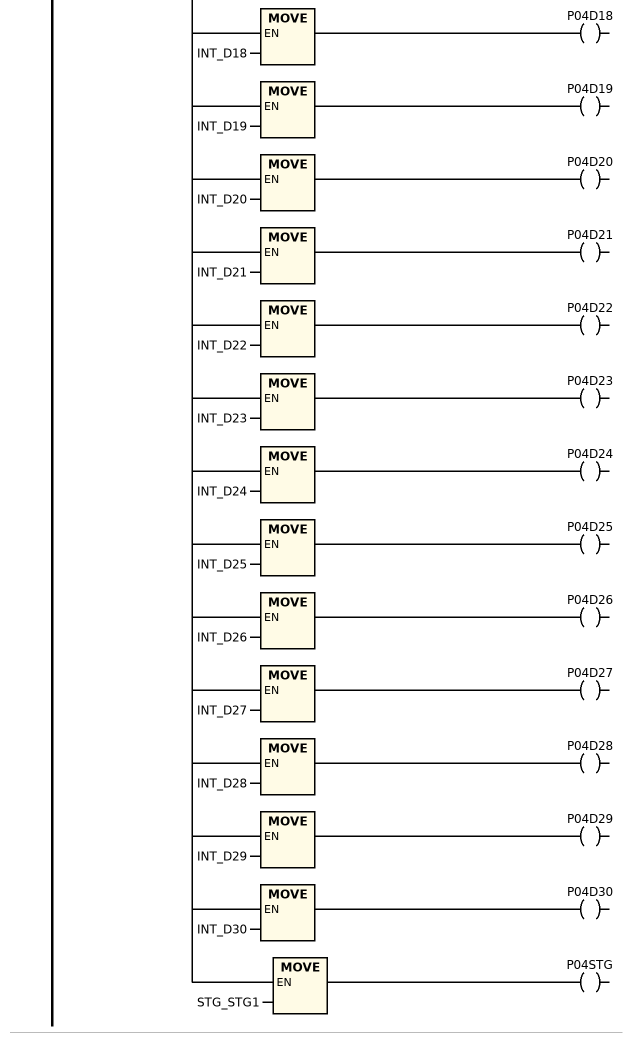
// NETWORK 25
_w134 := SV_HR AND P4B;
IF _w134 THEN _w135 := INT_D00; END_IF
P04D00 := _w135;
IF _w134 THEN _w136 := INT_D01; END_IF
P04D01 := _w136;
IF _w134 THEN _w137 := INT_D02; END_IF
P04D02 := _w137;
IF _w134 THEN _w138 := INT_D03; END_IF
P04D03 := _w138;
IF _w134 THEN _w139 := INT_D04; END_IF
P04D04 := _w139;
IF _w134 THEN _w140 := INT_D05; END_IF
P04D05 := _w140;
IF _w134 THEN _w141 := INT_D06; END_IF
P04D06 := _w141;
IF _w134 THEN _w142 := INT_D07; END_IF
P04D07 := _w142;
IF _w134 THEN _w143 := INT_D08; END_IF
P04D08 := _w143;
IF _w134 THEN _w144 := INT_D09; END_IF
P04D09 := _w144;
IF _w134 THEN _w145 := INT_D10; END_IF
P04D10 := _w145;
IF _w134 THEN _w146 := INT_D11; END_IF
P04D11 := _w146;
IF _w134 THEN _w147 := INT_D12; END_IF
P04D12 := _w147;
IF _w134 THEN _w148 := INT_D13; END_IF
P04D13 := _w148;
IF _w134 THEN _w149 := INT_D14; END_IF
P04D14 := _w149;
IF _w134 THEN _w150 := INT_D15; END_IF
P04D15 := _w150;
IF _w134 THEN _w151 := INT_D16; END_IF
P04D16 := _w151;
IF _w134 THEN _w152 := INT_D17; END_IF
P04D17 := _w152;
IF _w134 THEN _w153 := INT_D18; END_IF
P04D18 := _w153;
IF _w134 THEN _w154 := INT_D19; END_IF
P04D19 := _w154;
IF _w134 THEN _w155 := INT_D20; END_IF
P04D20 := _w155;
IF _w134 THEN _w156 := INT_D21; END_IF
P04D21 := _w156;
IF _w134 THEN _w157 := INT_D22; END_IF
P04D22 := _w157;
IF _w134 THEN _w158 := INT_D23; END_IF
P04D23 := _w158;
IF _w134 THEN _w159 := INT_D24; END_IF
P04D24 := _w159;
IF _w134 THEN _w160 := INT_D25; END_IF
P04D25 := _w160;
IF _w134 THEN _w161 := INT_D26; END_IF
P04D26 := _w161;
IF _w134 THEN _w162 := INT_D27; END_IF
P04D27 := _w162;
IF _w134 THEN _w163 := INT_D28; END_IF
P04D28 := _w163;
IF _w134 THEN _w164 := INT_D29; END_IF
P04D29 := _w164;
IF _w134 THEN _w165 := INT_D30; END_IF
P04D30 := _w165;
IF _w134 THEN _w166 := STG_STG1; END_IF
P04STG := _w166;

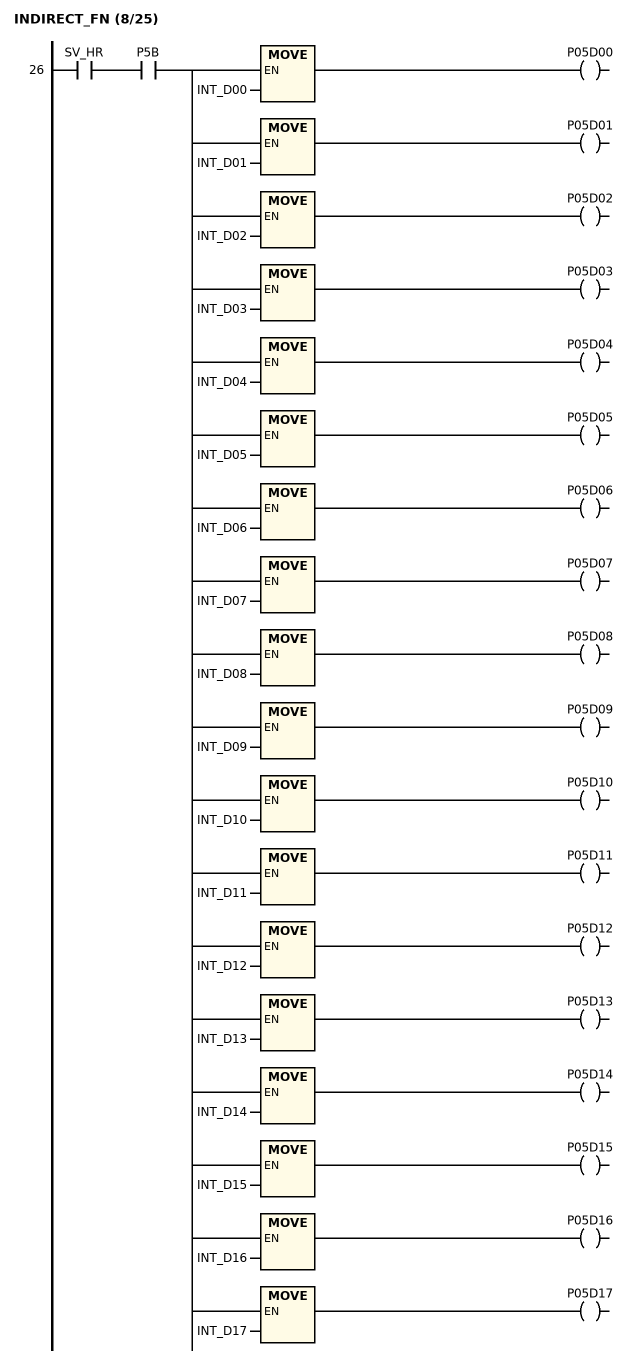
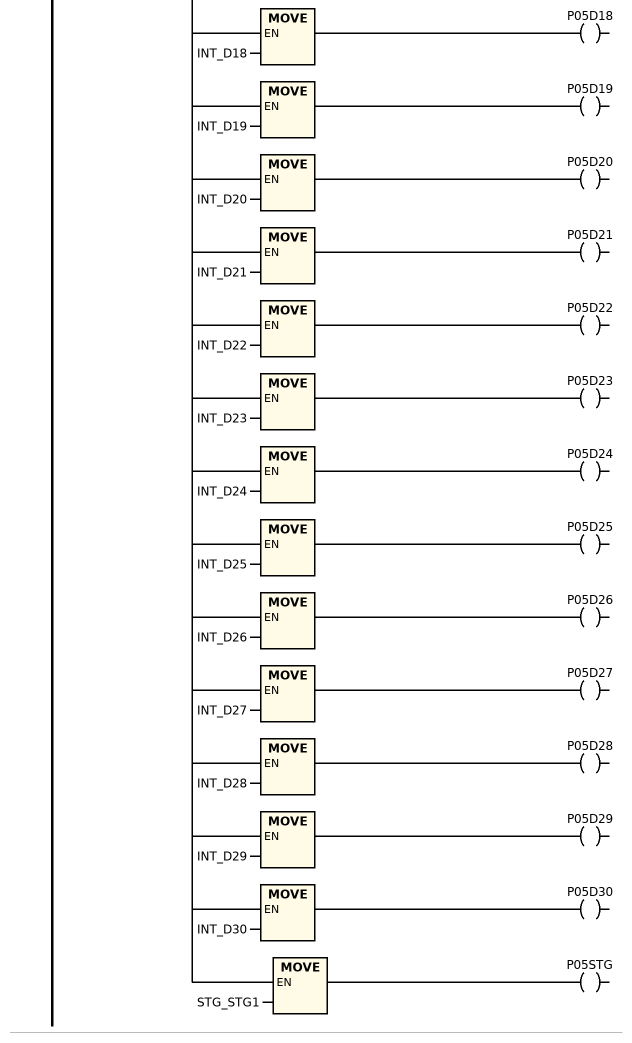
// NETWORK 26
_w167 := SV_HR AND P5B;
IF _w167 THEN _w168 := INT_D00; END_IF
P05D00 := _w168;
IF _w167 THEN _w169 := INT_D01; END_IF
P05D01 := _w169;
IF _w167 THEN _w170 := INT_D02; END_IF
P05D02 := _w170;
IF _w167 THEN _w171 := INT_D03; END_IF
P05D03 := _w171;
IF _w167 THEN _w172 := INT_D04; END_IF
P05D04 := _w172;
IF _w167 THEN _w173 := INT_D05; END_IF
P05D05 := _w173;
IF _w167 THEN _w174 := INT_D06; END_IF
P05D06 := _w174;
IF _w167 THEN _w175 := INT_D07; END_IF
P05D07 := _w175;
IF _w167 THEN _w176 := INT_D08; END_IF
P05D08 := _w176;
IF _w167 THEN _w177 := INT_D09; END_IF
P05D09 := _w177;
IF _w167 THEN _w178 := INT_D10; END_IF
P05D10 := _w178;
IF _w167 THEN _w179 := INT_D11; END_IF
P05D11 := _w179;
IF _w167 THEN _w180 := INT_D12; END_IF
P05D12 := _w180;
IF _w167 THEN _w181 := INT_D13; END_IF
P05D13 := _w181;
IF _w167 THEN _w182 := INT_D14; END_IF
P05D14 := _w182;
IF _w167 THEN _w183 := INT_D15; END_IF
P05D15 := _w183;
IF _w167 THEN _w184 := INT_D16; END_IF
P05D16 := _w184;
IF _w167 THEN _w185 := INT_D17; END_IF
P05D17 := _w185;
IF _w167 THEN _w186 := INT_D18; END_IF
P05D18 := _w186;
IF _w167 THEN _w187 := INT_D19; END_IF
P05D19 := _w187;
IF _w167 THEN _w188 := INT_D20; END_IF
P05D20 := _w188;
IF _w167 THEN _w189 := INT_D21; END_IF
P05D21 := _w189;
IF _w167 THEN _w190 := INT_D22; END_IF
P05D22 := _w190;
IF _w167 THEN _w191 := INT_D23; END_IF
P05D23 := _w191;
IF _w167 THEN _w192 := INT_D24; END_IF
P05D24 := _w192;
IF _w167 THEN _w193 := INT_D25; END_IF
P05D25 := _w193;
IF _w167 THEN _w194 := INT_D26; END_IF
P05D26 := _w194;
IF _w167 THEN _w195 := INT_D27; END_IF
P05D27 := _w195;
IF _w167 THEN _w196 := INT_D28; END_IF
P05D28 := _w196;
IF _w167 THEN _w197 := INT_D29; END_IF
P05D29 := _w197;
IF _w167 THEN _w198 := INT_D30; END_IF
P05D30 := _w198;
IF _w167 THEN _w199 := STG_STG1; END_IF
P05STG := _w199;

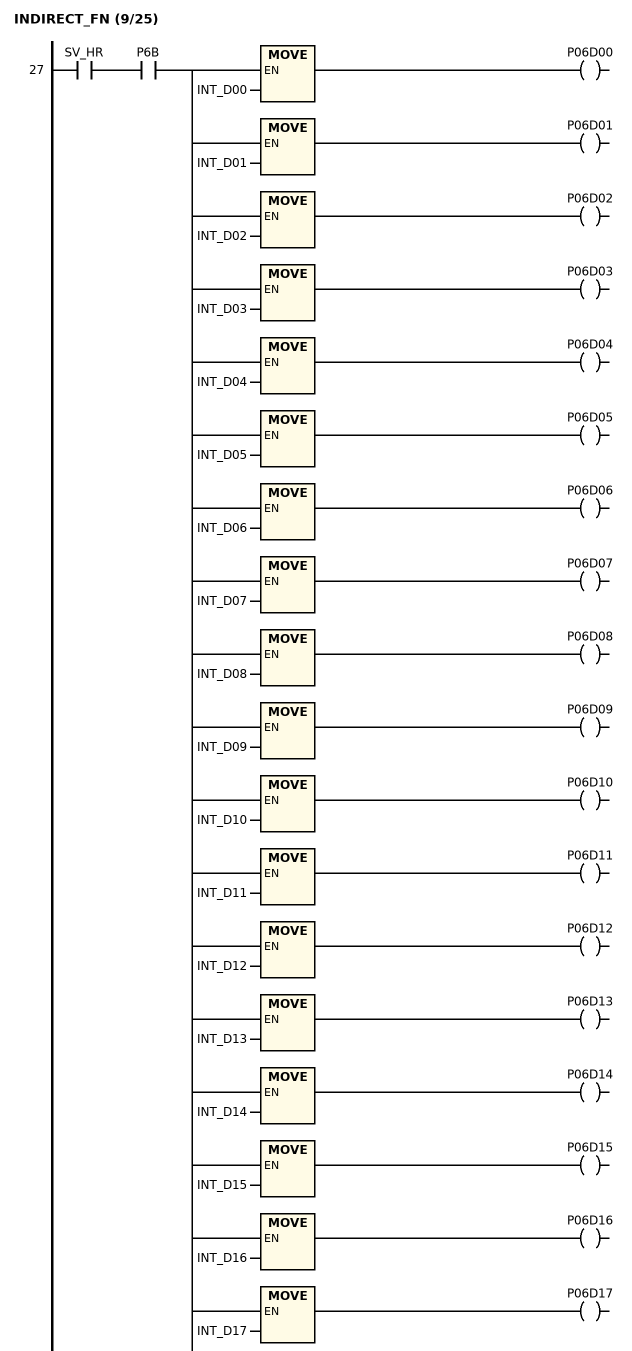
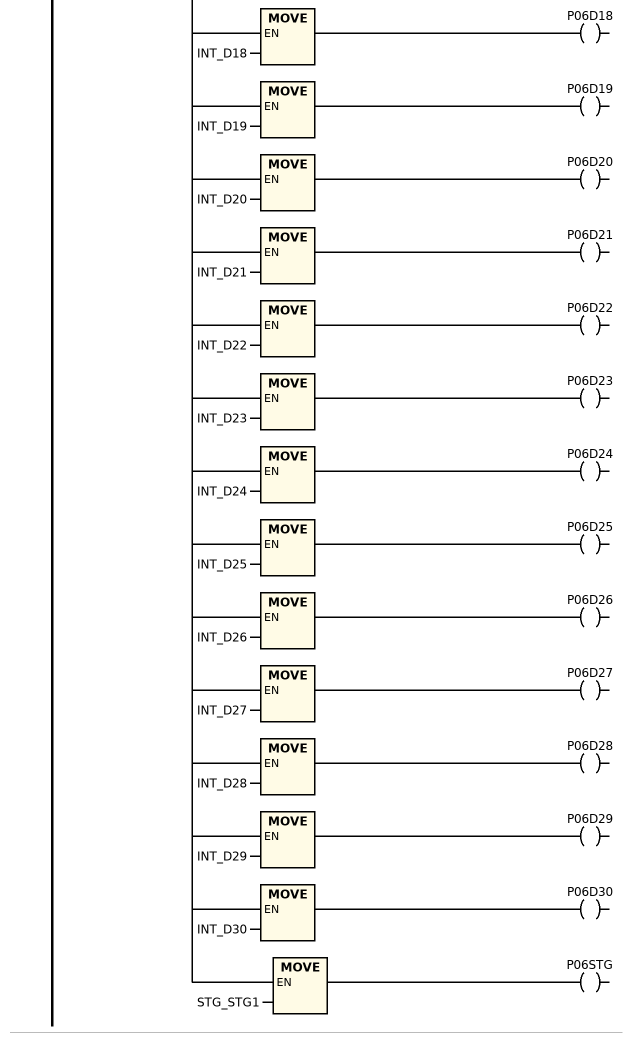
// NETWORK 27
_w200 := SV_HR AND P6B;
IF _w200 THEN _w201 := INT_D00; END_IF
P06D00 := _w201;
IF _w200 THEN _w202 := INT_D01; END_IF
P06D01 := _w202;
IF _w200 THEN _w203 := INT_D02; END_IF
P06D02 := _w203;
IF _w200 THEN _w204 := INT_D03; END_IF
P06D03 := _w204;
IF _w200 THEN _w205 := INT_D04; END_IF
P06D04 := _w205;
IF _w200 THEN _w206 := INT_D05; END_IF
P06D05 := _w206;
IF _w200 THEN _w207 := INT_D06; END_IF
P06D06 := _w207;
IF _w200 THEN _w208 := INT_D07; END_IF
P06D07 := _w208;
IF _w200 THEN _w209 := INT_D08; END_IF
P06D08 := _w209;
IF _w200 THEN _w210 := INT_D09; END_IF
P06D09 := _w210;
IF _w200 THEN _w211 := INT_D10; END_IF
P06D10 := _w211;
IF _w200 THEN _w212 := INT_D11; END_IF
P06D11 := _w212;
IF _w200 THEN _w213 := INT_D12; END_IF
P06D12 := _w213;
IF _w200 THEN _w214 := INT_D13; END_IF
P06D13 := _w214;
IF _w200 THEN _w215 := INT_D14; END_IF
P06D14 := _w215;
IF _w200 THEN _w216 := INT_D15; END_IF
P06D15 := _w216;
IF _w200 THEN _w217 := INT_D16; END_IF
P06D16 := _w217;
IF _w200 THEN _w218 := INT_D17; END_IF
P06D17 := _w218;
IF _w200 THEN _w219 := INT_D18; END_IF
P06D18 := _w219;
IF _w200 THEN _w220 := INT_D19; END_IF
P06D19 := _w220;
IF _w200 THEN _w221 := INT_D20; END_IF
P06D20 := _w221;
IF _w200 THEN _w222 := INT_D21; END_IF
P06D21 := _w222;
IF _w200 THEN _w223 := INT_D22; END_IF
P06D22 := _w223;
IF _w200 THEN _w224 := INT_D23; END_IF
P06D23 := _w224;
IF _w200 THEN _w225 := INT_D24; END_IF
P06D24 := _w225;
IF _w200 THEN _w226 := INT_D25; END_IF
P06D25 := _w226;
IF _w200 THEN _w227 := INT_D26; END_IF
P06D26 := _w227;
IF _w200 THEN _w228 := INT_D27; END_IF
P06D27 := _w228;
IF _w200 THEN _w229 := INT_D28; END_IF
P06D28 := _w229;
IF _w200 THEN _w230 := INT_D29; END_IF
P06D29 := _w230;
IF _w200 THEN _w231 := INT_D30; END_IF
P06D30 := _w231;
IF _w200 THEN _w232 := STG_STG1; END_IF
P06STG := _w232;

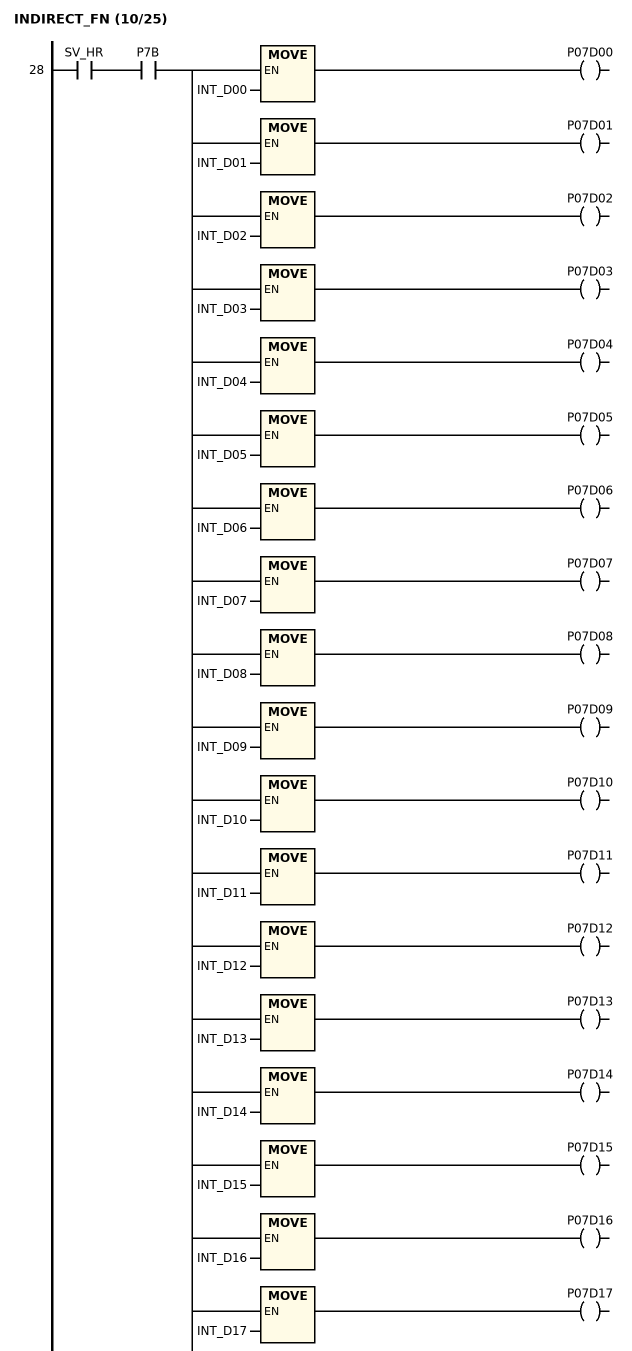
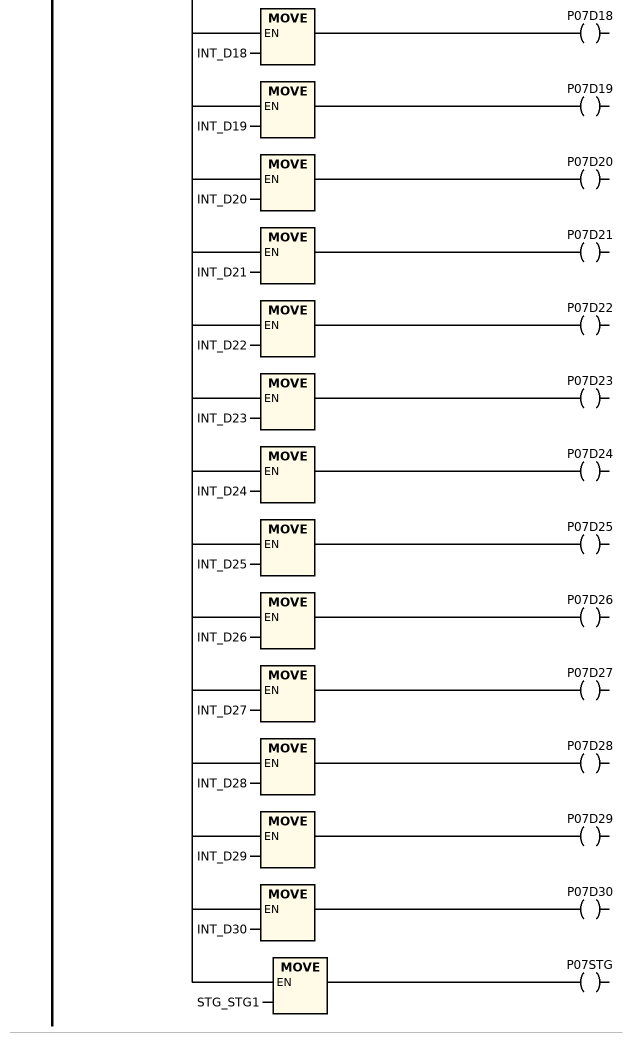
// NETWORK 28
_w233 := SV_HR AND P7B;
IF _w233 THEN _w234 := INT_D00; END_IF
P07D00 := _w234;
IF _w233 THEN _w235 := INT_D01; END_IF
P07D01 := _w235;
IF _w233 THEN _w236 := INT_D02; END_IF
P07D02 := _w236;
IF _w233 THEN _w237 := INT_D03; END_IF
P07D03 := _w237;
IF _w233 THEN _w238 := INT_D04; END_IF
P07D04 := _w238;
IF _w233 THEN _w239 := INT_D05; END_IF
P07D05 := _w239;
IF _w233 THEN _w240 := INT_D06; END_IF
P07D06 := _w240;
IF _w233 THEN _w241 := INT_D07; END_IF
P07D07 := _w241;
IF _w233 THEN _w242 := INT_D08; END_IF
P07D08 := _w242;
IF _w233 THEN _w243 := INT_D09; END_IF
P07D09 := _w243;
IF _w233 THEN _w244 := INT_D10; END_IF
P07D10 := _w244;
IF _w233 THEN _w245 := INT_D11; END_IF
P07D11 := _w245;
IF _w233 THEN _w246 := INT_D12; END_IF
P07D12 := _w246;
IF _w233 THEN _w247 := INT_D13; END_IF
P07D13 := _w247;
IF _w233 THEN _w248 := INT_D14; END_IF
P07D14 := _w248;
IF _w233 THEN _w249 := INT_D15; END_IF
P07D15 := _w249;
IF _w233 THEN _w250 := INT_D16; END_IF
P07D16 := _w250;
IF _w233 THEN _w251 := INT_D17; END_IF
P07D17 := _w251;
IF _w233 THEN _w252 := INT_D18; END_IF
P07D18 := _w252;
IF _w233 THEN _w253 := INT_D19; END_IF
P07D19 := _w253;
IF _w233 THEN _w254 := INT_D20; END_IF
P07D20 := _w254;
IF _w233 THEN _w255 := INT_D21; END_IF
P07D21 := _w255;
IF _w233 THEN _w256 := INT_D22; END_IF
P07D22 := _w256;
IF _w233 THEN _w257 := INT_D23; END_IF
P07D23 := _w257;
IF _w233 THEN _w258 := INT_D24; END_IF
P07D24 := _w258;
IF _w233 THEN _w259 := INT_D25; END_IF
P07D25 := _w259;
IF _w233 THEN _w260 := INT_D26; END_IF
P07D26 := _w260;
IF _w233 THEN _w261 := INT_D27; END_IF
P07D27 := _w261;
IF _w233 THEN _w262 := INT_D28; END_IF
P07D28 := _w262;
IF _w233 THEN _w263 := INT_D29; END_IF
P07D29 := _w263;
IF _w233 THEN _w264 := INT_D30; END_IF
P07D30 := _w264;
IF _w233 THEN _w265 := STG_STG1; END_IF
P07STG := _w265;

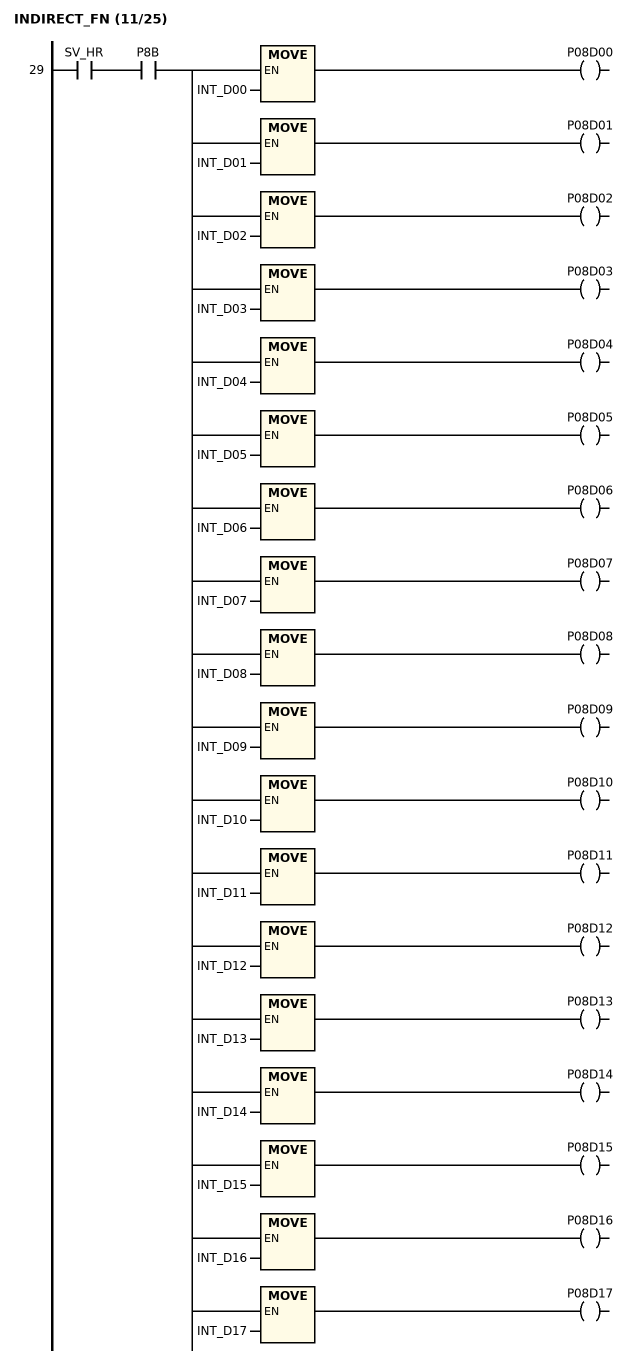
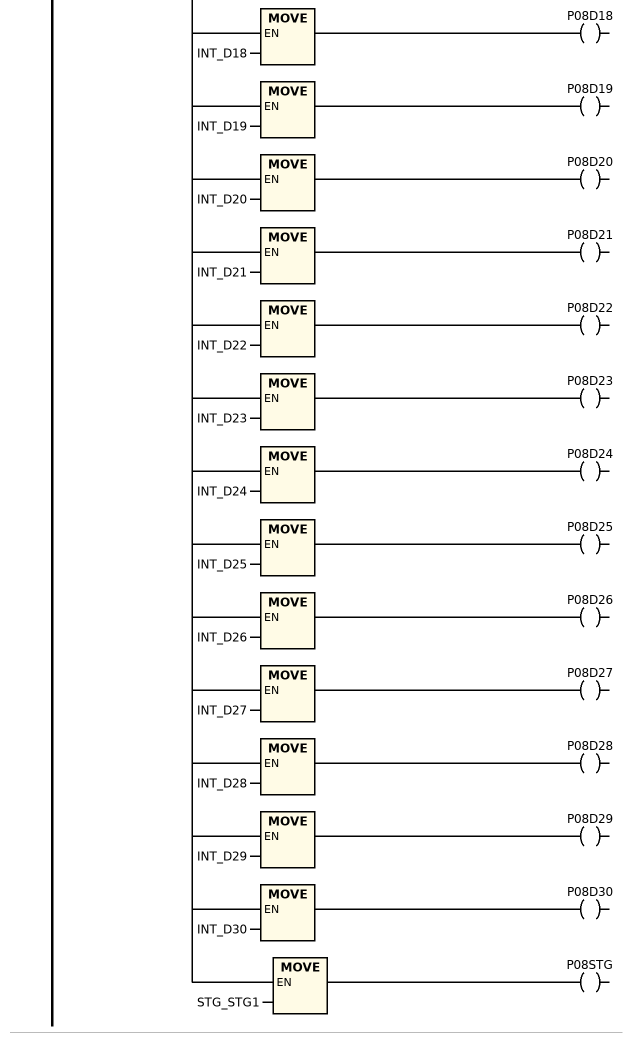
// NETWORK 29
_w266 := SV_HR AND P8B;
IF _w266 THEN _w267 := INT_D00; END_IF
P08D00 := _w267;
IF _w266 THEN _w268 := INT_D01; END_IF
P08D01 := _w268;
IF _w266 THEN _w269 := INT_D02; END_IF
P08D02 := _w269;
IF _w266 THEN _w270 := INT_D03; END_IF
P08D03 := _w270;
IF _w266 THEN _w271 := INT_D04; END_IF
P08D04 := _w271;
IF _w266 THEN _w272 := INT_D05; END_IF
P08D05 := _w272;
IF _w266 THEN _w273 := INT_D06; END_IF
P08D06 := _w273;
IF _w266 THEN _w274 := INT_D07; END_IF
P08D07 := _w274;
IF _w266 THEN _w275 := INT_D08; END_IF
P08D08 := _w275;
IF _w266 THEN _w276 := INT_D09; END_IF
P08D09 := _w276;
IF _w266 THEN _w277 := INT_D10; END_IF
P08D10 := _w277;
IF _w266 THEN _w278 := INT_D11; END_IF
P08D11 := _w278;
IF _w266 THEN _w279 := INT_D12; END_IF
P08D12 := _w279;
IF _w266 THEN _w280 := INT_D13; END_IF
P08D13 := _w280;
IF _w266 THEN _w281 := INT_D14; END_IF
P08D14 := _w281;
IF _w266 THEN _w282 := INT_D15; END_IF
P08D15 := _w282;
IF _w266 THEN _w283 := INT_D16; END_IF
P08D16 := _w283;
IF _w266 THEN _w284 := INT_D17; END_IF
P08D17 := _w284;
IF _w266 THEN _w285 := INT_D18; END_IF
P08D18 := _w285;
IF _w266 THEN _w286 := INT_D19; END_IF
P08D19 := _w286;
IF _w266 THEN _w287 := INT_D20; END_IF
P08D20 := _w287;
IF _w266 THEN _w288 := INT_D21; END_IF
P08D21 := _w288;
IF _w266 THEN _w289 := INT_D22; END_IF
P08D22 := _w289;
IF _w266 THEN _w290 := INT_D23; END_IF
P08D23 := _w290;
IF _w266 THEN _w291 := INT_D24; END_IF
P08D24 := _w291;
IF _w266 THEN _w292 := INT_D25; END_IF
P08D25 := _w292;
IF _w266 THEN _w293 := INT_D26; END_IF
P08D26 := _w293;
IF _w266 THEN _w294 := INT_D27; END_IF
P08D27 := _w294;
IF _w266 THEN _w295 := INT_D28; END_IF
P08D28 := _w295;
IF _w266 THEN _w296 := INT_D29; END_IF
P08D29 := _w296;
IF _w266 THEN _w297 := INT_D30; END_IF
P08D30 := _w297;
IF _w266 THEN _w298 := STG_STG1; END_IF
P08STG := _w298;

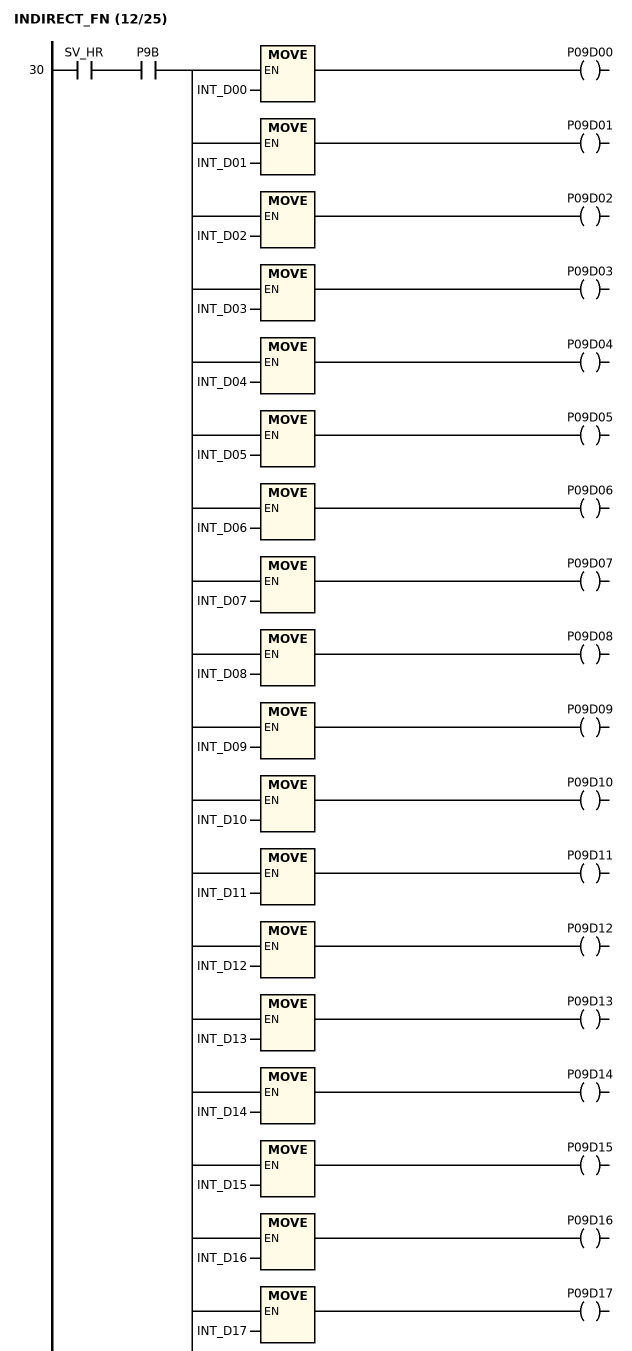
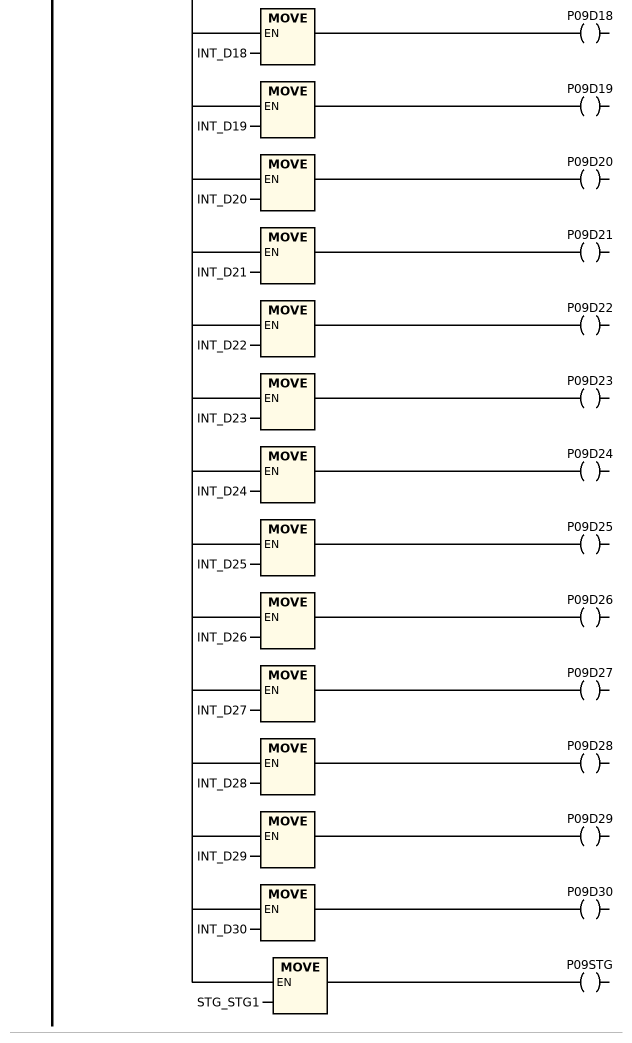
// NETWORK 30
_w299 := SV_HR AND P9B;
IF _w299 THEN _w300 := INT_D00; END_IF
P09D00 := _w300;
IF _w299 THEN _w301 := INT_D01; END_IF
P09D01 := _w301;
IF _w299 THEN _w302 := INT_D02; END_IF
P09D02 := _w302;
IF _w299 THEN _w303 := INT_D03; END_IF
P09D03 := _w303;
IF _w299 THEN _w304 := INT_D04; END_IF
P09D04 := _w304;
IF _w299 THEN _w305 := INT_D05; END_IF
P09D05 := _w305;
IF _w299 THEN _w306 := INT_D06; END_IF
P09D06 := _w306;
IF _w299 THEN _w307 := INT_D07; END_IF
P09D07 := _w307;
IF _w299 THEN _w308 := INT_D08; END_IF
P09D08 := _w308;
IF _w299 THEN _w309 := INT_D09; END_IF
P09D09 := _w309;
IF _w299 THEN _w310 := INT_D10; END_IF
P09D10 := _w310;
IF _w299 THEN _w311 := INT_D11; END_IF
P09D11 := _w311;
IF _w299 THEN _w312 := INT_D12; END_IF
P09D12 := _w312;
IF _w299 THEN _w313 := INT_D13; END_IF
P09D13 := _w313;
IF _w299 THEN _w314 := INT_D14; END_IF
P09D14 := _w314;
IF _w299 THEN _w315 := INT_D15; END_IF
P09D15 := _w315;
IF _w299 THEN _w316 := INT_D16; END_IF
P09D16 := _w316;
IF _w299 THEN _w317 := INT_D17; END_IF
P09D17 := _w317;
IF _w299 THEN _w318 := INT_D18; END_IF
P09D18 := _w318;
IF _w299 THEN _w319 := INT_D19; END_IF
P09D19 := _w319;
IF _w299 THEN _w320 := INT_D20; END_IF
P09D20 := _w320;
IF _w299 THEN _w321 := INT_D21; END_IF
P09D21 := _w321;
IF _w299 THEN _w322 := INT_D22; END_IF
P09D22 := _w322;
IF _w299 THEN _w323 := INT_D23; END_IF
P09D23 := _w323;
IF _w299 THEN _w324 := INT_D24; END_IF
P09D24 := _w324;
IF _w299 THEN _w325 := INT_D25; END_IF
P09D25 := _w325;
IF _w299 THEN _w326 := INT_D26; END_IF
P09D26 := _w326;
IF _w299 THEN _w327 := INT_D27; END_IF
P09D27 := _w327;
IF _w299 THEN _w328 := INT_D28; END_IF
P09D28 := _w328;
IF _w299 THEN _w329 := INT_D29; END_IF
P09D29 := _w329;
IF _w299 THEN _w330 := INT_D30; END_IF
P09D30 := _w330;
IF _w299 THEN _w331 := STG_STG1; END_IF
P09STG := _w331;

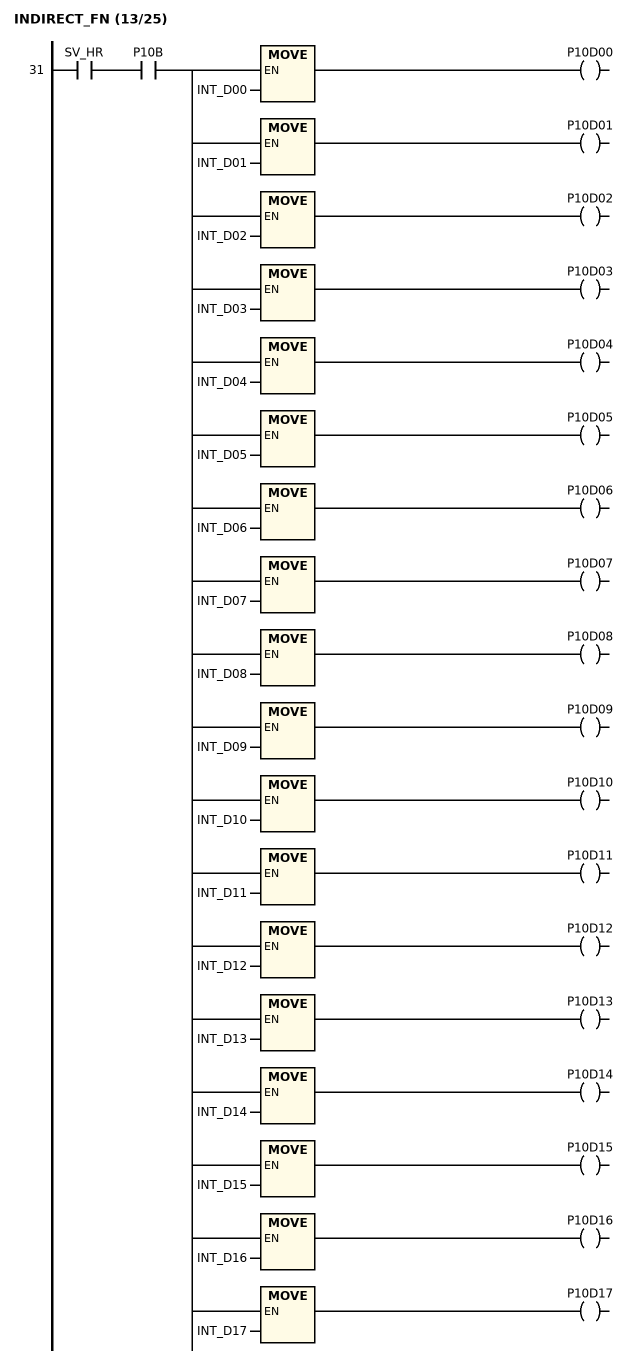
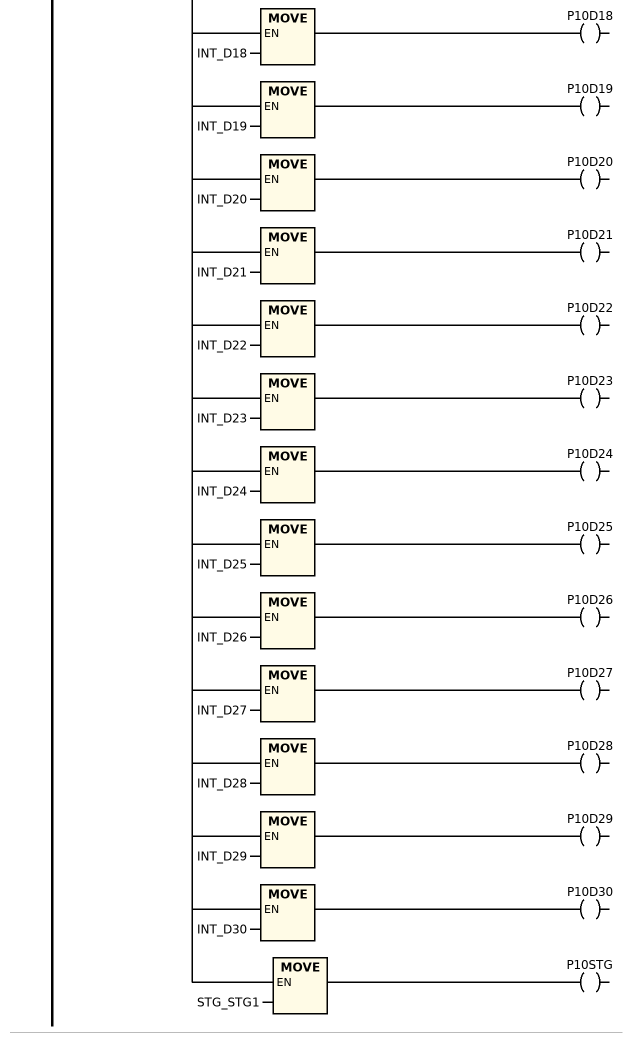
// NETWORK 31
_w332 := SV_HR AND P10B;
IF _w332 THEN _w333 := INT_D00; END_IF
P10D00 := _w333;
IF _w332 THEN _w334 := INT_D01; END_IF
P10D01 := _w334;
IF _w332 THEN _w335 := INT_D02; END_IF
P10D02 := _w335;
IF _w332 THEN _w336 := INT_D03; END_IF
P10D03 := _w336;
IF _w332 THEN _w337 := INT_D04; END_IF
P10D04 := _w337;
IF _w332 THEN _w338 := INT_D05; END_IF
P10D05 := _w338;
IF _w332 THEN _w339 := INT_D06; END_IF
P10D06 := _w339;
IF _w332 THEN _w340 := INT_D07; END_IF
P10D07 := _w340;
IF _w332 THEN _w341 := INT_D08; END_IF
P10D08 := _w341;
IF _w332 THEN _w342 := INT_D09; END_IF
P10D09 := _w342;
IF _w332 THEN _w343 := INT_D10; END_IF
P10D10 := _w343;
IF _w332 THEN _w344 := INT_D11; END_IF
P10D11 := _w344;
IF _w332 THEN _w345 := INT_D12; END_IF
P10D12 := _w345;
IF _w332 THEN _w346 := INT_D13; END_IF
P10D13 := _w346;
IF _w332 THEN _w347 := INT_D14; END_IF
P10D14 := _w347;
IF _w332 THEN _w348 := INT_D15; END_IF
P10D15 := _w348;
IF _w332 THEN _w349 := INT_D16; END_IF
P10D16 := _w349;
IF _w332 THEN _w350 := INT_D17; END_IF
P10D17 := _w350;
IF _w332 THEN _w351 := INT_D18; END_IF
P10D18 := _w351;
IF _w332 THEN _w352 := INT_D19; END_IF
P10D19 := _w352;
IF _w332 THEN _w353 := INT_D20; END_IF
P10D20 := _w353;
IF _w332 THEN _w354 := INT_D21; END_IF
P10D21 := _w354;
IF _w332 THEN _w355 := INT_D22; END_IF
P10D22 := _w355;
IF _w332 THEN _w356 := INT_D23; END_IF
P10D23 := _w356;
IF _w332 THEN _w357 := INT_D24; END_IF
P10D24 := _w357;
IF _w332 THEN _w358 := INT_D25; END_IF
P10D25 := _w358;
IF _w332 THEN _w359 := INT_D26; END_IF
P10D26 := _w359;
IF _w332 THEN _w360 := INT_D27; END_IF
P10D27 := _w360;
IF _w332 THEN _w361 := INT_D28; END_IF
P10D28 := _w361;
IF _w332 THEN _w362 := INT_D29; END_IF
P10D29 := _w362;
IF _w332 THEN _w363 := INT_D30; END_IF
P10D30 := _w363;
IF _w332 THEN _w364 := STG_STG1; END_IF
P10STG := _w364;

